FUNCTION_BLOCK "G297M_Code"	// FB 397
TITLE = G297M FAN KILN 2
//COPYRIGHT:    (C) 2009  BUHLER AG, CH-9240 UZWIL, SWITZERLAND
//
//PRODUCT:      WinCoS_BIW01_09
//
//TITLE:        FAN KILN 2
//                Machine group control
//                Maschinengruppensteuerung
// 
//--------------------------------------------------------------------------------
// 
//IDENT:        AUTHOR:             DEPT:                              DATE:
// 
//P01_FB397.2.0 M.Wedler            AEB41                              27.Apr.2010
//             2nd Release
//P01_FB397.1.0 K.Renz              CSB41                              06.Nov.2009
//             1st Release
// 
//--------------------------------------------------------------------------------
// 
//PURPOSE: 
// 
//MANUAL : 
// 
//RESTRICTIONS: 
// 
//--------------------------------------------------------------------------------
//
AUTHOR : KR
FAMILY : USW
VERSION : 9.9
VAR
  Gr : FB 10;	//Standard interface to group
  InOutValue1 : DINT ;	//Data for user
  InOutValue2 : DINT ;	//Data for user
  OutWayConflict : BOOL ;	//Data for user
  OutSelectionOk : BOOL ;	//Data for user
  CmdNewValue : BOOL ;	//Data for user
  CmdNewJob : BOOL ;	//Data for user
  OutCodeOK : BOOL ;	//Data for user
  InEndOfJob : BOOL ;	//Data for user
  staWayOk : BOOL ;	//Data for user
  EdgeStartRelease : BOOL ;	//Data for user
  USW8 : BOOL ;	//Data for user
  USW9 : BOOL ;	//Data for user
  USW10 : BOOL ;	//Data for user
  USW11 : BOOL ;	//Data for user
  USW12 : BOOL ;	//Data for user
  USW13 : BOOL ;	//Data for user
  USW14 : BOOL ;	//Data for user
  USW15 : BOOL ;	//Data for user
  A_3225_KCU04AI1 : FB 19;	// AnaInp
  A_3225_KCU04AI2 : FB 19;	// AnaInp
  A_3225_BTE05 : FB 19;	// AnaInp
  A_3225_BTE06 : FB 19;	// AnaInp
  A_3225_TSC01 : FB 14;	// DigInpCont
  A_3225_MXZ01MA : FB 1032;	// Motor+6DI
  A_3225_TSC01_AC : FB 19;	// AnaInp
  A_3225_TSC01_AF : FB 19;	// AnaInp
  A_3225_TSC01_AP : FB 19;	// AnaInp
  A_3225_TSC01_AT : FB 19;	// AnaInp
  A_3225_TSC01_COM : FB 1816;	// FU_Siemens
  A_3226_KCU04AI1 : FB 19;	// AnaInp
  A_3226_KCU04AI2 : FB 19;	// AnaInp
  A_3226_BTE05 : FB 19;	// AnaInp
  A_3226_BTE06 : FB 19;	// AnaInp
  A_3226_MXZ01MA : FB 1033;	// Motor+6DI
  A_3226_TSC01_AC : FB 19;	// AnaInp
  A_3226_TSC01_AF : FB 19;	// AnaInp
  A_3226_TSC01_AP : FB 19;	// AnaInp
  A_3226_TSC01_AT : FB 19;	// AnaInp
  A_3226_TSC01_COM : FB 1816;	// FU_Siemens
  A_3226_TSC01 : FB 14;	// DigInpCont
END_VAR
VAR_TEMP
  tmpEnable : BOOL ;
  tmpFlag : BOOL ;
  tmpCmdNext : BOOL ;
  tmpLocal : BOOL ;
  tmpAspOk : BOOL ;
  tmpHWStop : BOOL ;
  tmpInstanzDBNo : INT ;
END_VAR
BEGIN
NETWORK
TITLE =
NETWORK
TITLE = Read command from group control
//Parameter
      SET;
      S     DB9.DBX 87.0;
      R     DB9.DBX 127.0;
      R     DB9.DBX 167.0;
      R     DB9.DBX 47.0;
      R     DB9.DBX 207.0;
      S     DIX [AR2,P#32.0];
      R     DIX [AR2,P#32.1];
      R     DIX [AR2,P#32.2];
//Command
      A     DB9.DBX 327.0;
      =     DIX [AR2,P#14.0];
      A     DB9.DBX 287.0;
      =     DIX [AR2,P#15.4];
      A     DB9.DBX 407.0;
      R     DB9.DBX 407.0;
      S     DIX [AR2,P#15.3];
      A     DB9.DBX 367.0;
      R     DB9.DBX 367.0;
      S     DIX [AR2,P#15.2];
      A     DB9.DBX 447.0;
      AN    DIX [AR2,P#15.5];
      S     DIX [AR2,P#14.7];
      A     DB9.DBX 447.0;
      R     DB9.DBX 447.0;
//      U     "GCS7_GrCtrlDB".CmdManualOff[297]
//      O     "GCS7_GrCtrlDB".OutOccupied[297]
//      R     "GCS7_GrCtrlDB".CmdManualOff[297]
//      S     #Gr.CmdManualOff
      A     DB9.DBX 767.0;
      R     DB9.DBX 767.0;
      S     DIX [AR2,P#14.1];
//Init Line Number
      A     DB9.DBX 207.0;
      JCN   WE00;
      L     0;
      T     DIW [AR2,P#24.0];
WE00: NOP   0;
NETWORK
TITLE = Call Methode Control
// 1. Handle Interface PCControl      
// 2. Prepare mode --> ModePassive,ModeActive,ModeIdling      
// 3. Reset global flags of the group
      BLD   14;
      =     L 10.0;
      L     DINO;
      T     LW 8;
      CDB;
      OPN   DI [LW 8];
      TAR2  LD 4;
      L     1;
      T     DIW [AR2,P#0.0];
      +AR2  P#0.0;
      UC    FB 10;
      LAR2  LD 4;
      CDB;
      BLD   15;
NETWORK
TITLE = Restart Idling Time
      L     DIW [AR2,P#36.0];
      L     2;
      >=I;
      JC    IdTm;
      T     DIW [AR2,P#36.0];
IdTm: NOP   0;
      CLR;
      S     DIX [AR2,P#14.2];
NETWORK
TITLE = Prepare global flags
NETWORK
TITLE = Set Pattern (Target position)
      A     DIX [AR2,P#15.5];
      JC    ILO6;
// Drehzahlabsenkung wenn die andere Horde im Cooling ist
// und die Temperatur unter der eigenen Horde 5°C > als T[Soll] 
//      U     "MAL1S032Par".Par.FlagProcess.Cooling_Activ
//      U     "G302M".USW8                // Temperatur unter der Horde 5°C > T[Soll]
//      L     50                          // 50%
//      SPB   En06
      L     DB922.DBW 228;
//      U     "G275M".USW8                // Drehzahlverrinderung bei offenen Bypassklappen
//      SPBN  En06
//      L     DB799.DBW   26              // Sollwert vom LS
//      -I    
      JU    En06;
ILO6: NOP   0;
      L     DB923.DBW 284;
En06: NOP   0;
      L     100;
      *I;
      T     DIW [AR2,P#1052.0];	// xxx.xx%
      T     DIW [AR2,P#2046.0];	// xxx.xx%
NETWORK
TITLE = Interlocking WayOk
NETWORK
TITLE = Interlocking Autostart
      CLR;
      R     DIX [AR2,P#18.4];
NETWORK
TITLE = Interlocking Enable
// (network holds code this reader does not know; not shown)
//--------------------- Ein-Hordenbetrieb ----------------------------//
// Luft-Eintritt
// Luft-Austritt
//---------------------- Zwei-Hordenbetrieb --------------------------//
// Luft-Eintritt
//MW 2010.04.29      U     "G273M".A_3135_MXZ11.StHN   // Louver Air Heater Kilningbox 1
//MW 2010.04.29      U     "G299M".A_3236_MXZ11.StHN   // Recycling Air Flap Kilningbox 2
// Luft-Austritt
//MW 2010.04.29      U     "G299M".A_3235_MXZ11.StHN   // Recycling Air Flap Kilningbox 2
//MW 2010.04.29      UN    "G299M".A_3236_MXZ11.StLN   // Recycling Air Flap Kilningbox 2
//MW 2010.04.29      UN    "G273M".A_3136_MXZ11.StLN   // Recycling Air Flap Kilningbox 1
// 100% Umluft-Betrieb
//MW 2010.04.29      U     "G299M".A_3235_MXZ11.StHN   // Recycling Air Flap Kilningbox 2
//MW 2010.04.29      O     "G273M".A_3136_MXZ11.StHN   // Recycling Air Flap Kilningbox 1
//MW 2010.04.29      O     "G299M".A_3236_MXZ11.StHN   // Recycling Air Flap Kilningbox 2
NETWORK
TITLE = Interlocking Next
      A     DIX [AR2,P#15.2];
      A     DIX [AR2,P#18.4];
      AN    DIX [AR2,P#19.6];
      =     #tmpCmdNext;
NETWORK
TITLE = Interlocking Local / HWStop
      A     DB50.DBX 32.4;
      =     #tmpHWStop;
      A     DIX [AR2,P#16.0];
      O     #tmpHWStop;
      =     #tmpLocal;
NETWORK
TITLE = Interlocking Start Warning
      NOP   0;
//- Restart after fault --
      A     DIX [AR2,P#15.3];
      A     DIX [AR2,P#19.2];
      S     DB100.DBX 136.4;
//- Run Timer --
      OPN   "G297M";
      CALL  FB 100 , DB 100 (
           DIX 0.0                  := FALSE,
           DIW 2                    := 11,
           DIX 4.0                  := DBX [AR2,P#18.0],
           DIX 4.1                  := #tmpLocal,
           DIX 4.2                  := DBX [AR2,P#19.1],
           DIX 4.3                  := #tmpCmdNext,
           DIX 6.0                  := #tmpCmdNext,
           DIX 6.1                  := DBX [AR2,P#19.3]);
//- Store Startwarning done  --
//- Reset Autostart --
      A     DB100.DBX 236.1;
      FN    DIX [AR2,P#58.7];
      A     DIX [AR2,P#19.2];
      R     DIX [AR2,P#18.4];
NETWORK
TITLE = =A-3225-KCU04AI1 : VIBRATION MONITOR FAN 1 CHANNEL 1
//Alarm Level = 10.00mm/sec
//Trip Level = 11.20mm/sec
      NOP   0;
//-InLocal---
      A     #tmpLocal;
      O     DB923.DBX 1569.0;	// emergency regime without fan 1
      =     DIX [AR2,P#63.4];
//-Monitoring--- 
      CLR;
      =     DIX [AR2,P#62.0];
      CLR;
      =     DIX [AR2,P#62.1];
      CLR;
      =     DIX [AR2,P#62.2];
      SET;
      =     DIX [AR2,P#62.3];
      SET;
      =     DIX [AR2,P#62.4];
// 
//-Read inputs---
      L     PIW 1054;
      L     0;
      <I;
      JC    v003;
      TAK;
v003: T     DIW [AR2,P#66.0];
      A     DB50.DBX 32.4;
      =     DIX [AR2,P#63.0];
      A     DB51.DBX 12.5;
      =     DIX [AR2,P#63.1];
// 
//-Set Parameters---
// --> Erläuterung
      L     L#2540;	// 20mA = 25.40mm/sec       
      T     DB397.DBD 90;
      L     L#10000;	// OutValuePc=OutValueUnits
      T     DB397.DBD 94;
      L     L#-1;	// -0.01mm/sec
      T     DB397.DBD 98;
      L     L#0;	// 0.00mm/sec
      T     DB397.DBD 102;
      L     L#1000;	// 10.00mm/sec
      T     DB397.DBD 106;
      L     L#1120;	// 11.20mm/sec
      T     DB397.DBD 110;
      SET;
      =     DB397.DBX 84.6;
      =     DB397.DBX 84.7;
      =     DB397.DBX 85.0;
      =     DB397.DBX 85.1;
      =     DB397.DBX 85.6;
      =     DB397.DBX 85.7;
      CLR;
      =     DB397.DBX 85.2;
// 
//-Call object control---
      BLD   14;
// 
//-Write outputs---
      =     L 10.0;
      L     DINO;
      T     LW 8;
      CDB;
      OPN   DI [LW 8];
      TAR2  LD 4;
      +AR2  P#60.0;
      UC    FB 19;
      LAR2  LD 4;
      CDB;
      BLD   15;
NETWORK
TITLE = =A-3225-KCU04AI2 : VIBRATION MONITOR FAN 1 CHANNEL 2
//Alarm Level = 10.00mm/sec
//Trip Level = 11.20mm/sec
      NOP   0;
//-InLocal---
      A     #tmpLocal;
      O     DB923.DBX 1569.0;	// emergency regime without fan 1
      =     DIX [AR2,P#151.4];
//-Monitoring--- 
      CLR;
      =     DIX [AR2,P#150.0];
      CLR;
      =     DIX [AR2,P#150.1];
      CLR;
      =     DIX [AR2,P#150.2];
      SET;
      =     DIX [AR2,P#150.3];
      SET;
      =     DIX [AR2,P#150.4];
// 
//-Read inputs---
      L     PIW 1052;
      L     0;
      <I;
      JC    v004;
      TAK;
v004: T     DIW [AR2,P#154.0];
      A     DB50.DBX 32.4;
      =     DIX [AR2,P#151.0];
      A     DB51.DBX 12.5;
      =     DIX [AR2,P#151.1];
// 
//-Set Parameters---
// --> Erläuterung
      L     L#2540;	// 20mA = 25.40mm/sec       
      T     DB397.DBD 178;
      L     L#10000;	// OutValuePc=OutValueUnits
      T     DB397.DBD 182;
      L     L#-1;	// -0.01mm/sec
      T     DB397.DBD 186;
      L     L#0;	// 0.00mm/sec
      T     DB397.DBD 190;
      L     L#1000;	// 10.00mm/sec
      T     DB397.DBD 194;
      L     L#1120;	// 11.20mm/sec
      T     DB397.DBD 198;
      SET;
      =     DB397.DBX 172.6;
      =     DB397.DBX 172.7;
      =     DB397.DBX 173.0;
      =     DB397.DBX 173.1;
      =     DB397.DBX 173.6;
      =     DB397.DBX 173.7;
      CLR;
      =     DB397.DBX 173.2;
// 
//-Call object control---
      BLD   14;
// 
//-Write outputs---
      =     L 10.0;
      L     DINO;
      T     LW 8;
      CDB;
      OPN   DI [LW 8];
      TAR2  LD 4;
      +AR2  P#148.0;
      UC    FB 19;
      LAR2  LD 4;
      CDB;
      BLD   15;
NETWORK
TITLE = =A-3225-BTE05 : TEMPERATURE BEARING TEMPERATUR SENSOR
//Alarm Level = 100.00°C    
//Trip Level = 110.00°C
      NOP   0;
//-InLocal---
      A     #tmpLocal;
      O     DB923.DBX 1569.0;	// emergency regime without fan 1
      =     DIX [AR2,P#239.4];
//-Monitoring--- 
      CLR;
      =     DIX [AR2,P#238.0];
      CLR;
      =     DIX [AR2,P#238.1];
      CLR;
      =     DIX [AR2,P#238.2];
      SET;
      =     DIX [AR2,P#238.3];
      SET;
      =     DIX [AR2,P#238.4];
// 
//-Read inputs---
      L     PIW 1028;
      T     DIW [AR2,P#242.0];
      A     DB50.DBX 32.4;
      =     DIX [AR2,P#239.0];
      A     DB51.DBX 12.5;
      =     DIX [AR2,P#239.1];
//To Block Problems with Sensor
      L     600;
      T     DB397.DBW 296;
      T     DB397.DBW 298;
// 
//-Set Parameters---
// --> Erläuterung
      L     L#27648;	// Temperature direkt      
      T     DB397.DBD 266;
      L     L#10000;	// OutValuePc=OutValueUnits
      T     DB397.DBD 270;
      L     L#0;	// 0.00°C
      T     DB397.DBD 274;
      L     L#100;	// 1.00°C
      T     DB397.DBD 278;
      L     L#10000;	// 100.00°C
      T     DB397.DBD 282;
      L     L#11000;	// 110.00°C
      T     DB397.DBD 286;
      SET;
      =     DB397.DBX 260.6;
      =     DB397.DBX 260.7;
      =     DB397.DBX 261.0;
      =     DB397.DBX 261.1;
      =     DB397.DBX 261.6;
      =     DB397.DBX 261.7;
      CLR;
      =     DB397.DBX 261.2;
// 
//-Call object control---
      BLD   14;
// 
//-Write outputs---
      =     L 10.0;
      L     DINO;
      T     LW 8;
      CDB;
      OPN   DI [LW 8];
      TAR2  LD 4;
      +AR2  P#236.0;
      UC    FB 19;
      LAR2  LD 4;
      CDB;
      BLD   15;
NETWORK
TITLE = =A-3225-BTE06 : TEMPERATURE BEARING TEMPERATUR SENSOR
//Alarm Level = 100.00°C    
//Trip Level = 110.00°C
      NOP   0;
//-InLocal---
      A     #tmpLocal;
      O     DB923.DBX 1569.0;	// emergency regime without fan 1
      =     DIX [AR2,P#327.4];
//-Monitoring--- 
      SET;
      =     DIX [AR2,P#326.0];
      CLR;
      =     DIX [AR2,P#326.1];
      CLR;
      =     DIX [AR2,P#326.2];
      SET;
      =     DIX [AR2,P#326.3];
      SET;
      =     DIX [AR2,P#326.4];
// 
//-Read inputs---
      L     PIW 1030;
      T     DIW [AR2,P#330.0];
      A     DB50.DBX 32.4;
      =     DIX [AR2,P#327.0];
      A     DB51.DBX 12.5;
      =     DIX [AR2,P#327.1];
//To Block Problems with Sensor
      L     600;
      T     DB397.DBW 384;
      T     DB397.DBW 386;
// 
//-Set Parameters---
// --> Erläuterung
      L     L#27648;	// Temperature direkt      
      T     DB397.DBD 354;
      L     L#10000;	// OutValuePc=OutValueUnits
      T     DB397.DBD 358;
      L     L#0;	// 0.00°C
      T     DB397.DBD 362;
      L     L#100;	// 1.00°C
      T     DB397.DBD 366;
      L     L#10000;	// 100.00°C
      T     DB397.DBD 370;
      L     L#11000;	// 110.00°C
      T     DB397.DBD 374;
      SET;
      =     DB397.DBX 348.6;
      =     DB397.DBX 348.7;
      =     DB397.DBX 349.0;
      =     DB397.DBX 349.1;
      =     DB397.DBX 349.6;
      =     DB397.DBX 349.7;
      CLR;
      =     DB397.DBX 349.2;
// 
//-Call object control---
      BLD   14;
// 
//-Write outputs---
      =     L 10.0;
      L     DINO;
      T     LW 8;
      CDB;
      OPN   DI [LW 8];
      TAR2  LD 4;
      +AR2  P#324.0;
      UC    FB 19;
      LAR2  LD 4;
      CDB;
      BLD   15;
NETWORK
TITLE = =A-3225-MXZ01MA : FAN 1
      NOP   0;
//-InLocal---
      A     #tmpLocal;
      O     DB923.DBX 1569.0;	// emergency regime without fan 1
      =     DIX [AR2,P#449.4];
//-Interlocking---
      AN    DB923.DBX 1569.0;	// emergency regime without fan 1
      A(;
      AN    DIX [AR2,P#1445.4];
      O     DB923.DBX 1569.1;	// emergency regime without fan 2
      );
      A(;
      A     DIX [AR2,P#15.5];
      A     DIX [AR2,P#14.5];
      ON    DIX [AR2,P#15.5];
      );
      AN    DIX [AR2,P#65.7];	// Vibrationswächter 1
      AN    DIX [AR2,P#153.7];	// Vibrationswächter 2
      AN    DIX [AR2,P#241.7];	// Lager Temperatur 1
      AN    DIX [AR2,P#329.7];	// Lager Temperatur 2
      AN    DB376.DBX 65.4;	// Differenzdruck hinter dem Waermetauscher
      A     DIX [AR2,P#18.0];
      =     DIX [AR2,P#448.1];
      A     #tmpCmdNext;
//      U     "MAL1S033Par".Par.FlagProcess2.Schaltp_5
      S     DIX [AR2,P#449.2];
      A     DIX [AR2,P#19.7];
      =     DIX [AR2,P#449.7];
// 
//=Values and commands of elements===
//-=A-3225-KCU04---
//      CLR
//      S     #A_3225_MXZ01MA.A_3225_KCU04.CmdRunTimeOutTime
//-=A-3225-MXZ01_SM---
//      CLR
//      S     #A_3225_MXZ01MA.A_3225_MXZ01_SM.CmdRunTimeOutTime
// 
//-Read inputs of elements---
      O     DIX [AR2,P#451.1];
      O     DIX [AR2,P#451.2];
      =     DIX [AR2,P#494.6];
      A     I 1026.6;
      =     DIX [AR2,P#460.6];
      A     DB50.DBX 32.4;
      =     DIX [AR2,P#462.0];
      A     DB51.DBX 12.6;
      =     DIX [AR2,P#462.1];
      A     DB50.DBX 32.4;
      =     DIX [AR2,P#496.0];
      A     DIX [AR2,P#1050.4];
      O     DB50.DBX 33.0;
      A     DIX [AR2,P#666.6];
      =     DIX [AR2,P#664.6];
      A     DB50.DBX 32.4;
      =     DIX [AR2,P#666.0];
// Überwachung Profibus-Kommunikation
      A     DB51.DBX 12.7;	// FU  ?????
      =     DIX [AR2,P#666.1];
// 
//-Set Parameters---
// 
//-Call object control---
      BLD   14;
// 
//-Write outputs---
      =     L 10.0;
      L     DINO;
      T     LW 8;
      CDB;
      OPN   DI [LW 8];
      TAR2  LD 4;
      +AR2  P#446.0;
      UC    "A_3225_MXZ01MA_Code";
      LAR2  LD 4;
      CDB;
      BLD   15;
NETWORK
TITLE = =A-3225-TSC01_COM : FAN 1 FU KOMMUNIKATION
      NOP   0;
      A     DIX [AR2,P#666.6];
      =     DIX [AR2,P#1050.1];
//      U     #A_3225_MXZ01MA.A_3225_MXZ01.OutpRunRev
      CLR;
      =     DIX [AR2,P#1050.0];
      A     DIX [AR2,P#15.3];
      O     DIX [AR2,P#462.6];
      S     DIX [AR2,P#1050.2];
// 
//-Read inputs---
// 
//-Set Parameters---
// 
//-Call object control---
      BLD   14;
// 
//-Write outputs---
      =     L 10.0;
      L     DINO;
      T     LW 8;
      CDB;
      OPN   DI [LW 8];
      TAR2  LD 4;
      +AR2  P#1048.0;
      UC    FB 1816;
      LAR2  LD 4;
      CDB;
      BLD   15;
NETWORK
TITLE = =A-3225-TSC01_AC : ACT. CURRENT FAN 1 FU 
//20000Dez=100,0%=720,0A
//Analog Input 20mA=27648Dez=995,3A
      NOP   0;
//-InLocal---
      A     #tmpLocal;
      O     DB923.DBX 1569.0;	// emergency regime without fan 1
      =     DIX [AR2,P#699.4];
//-Monitoring--- 
      SET;
      =     DIX [AR2,P#698.0];
      CLR;
      =     DIX [AR2,P#698.1];
      CLR;
      =     DIX [AR2,P#698.2];
      CLR;
      =     DIX [AR2,P#698.3];
      CLR;
      =     DIX [AR2,P#698.4];
// 
//-Read inputs---
      L     DIW [AR2,P#1058.0];
      T     DIW [AR2,P#702.0];
      A     DB50.DBX 32.4;
      =     DIX [AR2,P#699.0];
// 
//-Set Parameters---
// --> Erläuterung
      L     L#9953;	// Stromwert bei 27648Dez
      T     DB397.DBD 726;
      L     L#10000;	// OutValuePc=OutValueUnits
      T     DB397.DBD 730;
      L     L#0;	// 0.0A
      T     DB397.DBD 734;
      L     L#4000;	// 40.0A
      T     DB397.DBD 738;
      L     L#7200;	// 720.0A=100.0%
      T     DB397.DBD 742;
      L     L#9360;	// 936.0A=130.0%
      T     DB397.DBD 746;
// 
//-Call object control---
      BLD   14;
// 
//-Write outputs---
      =     L 10.0;
      L     DINO;
      T     LW 8;
      CDB;
      OPN   DI [LW 8];
      TAR2  LD 4;
      +AR2  P#696.0;
      UC    FB 19;
      LAR2  LD 4;
      CDB;
      BLD   15;
NETWORK
TITLE = =A-3225-TSC01_AF : ACT. FREQUENCY FAN 1 FU 
      NOP   0;
//-InLocal---
      A     #tmpLocal;
      O     DB923.DBX 1569.0;	// emergency regime without fan 1
      =     DIX [AR2,P#787.4];
//-Monitoring--- 
      SET;
      =     DIX [AR2,P#786.0];
      CLR;
      =     DIX [AR2,P#786.1];
      CLR;
      =     DIX [AR2,P#786.2];
      CLR;
      =     DIX [AR2,P#786.3];
      CLR;
      =     DIX [AR2,P#786.4];
// 
//-Read inputs---
      L     DIW [AR2,P#1048.0];	// Umgerechnet in FU-FB
      T     DIW [AR2,P#790.0];
      A     DB50.DBX 32.4;
      =     DIX [AR2,P#787.0];
// 
//-Set Parameters---
// --> Erläuterung
      L     L#27648;	// InpValue=Drehzahl direkt   
      T     DB397.DBD 814;
      L     L#10000;	// OutValuePc=OutValueUnits
      T     DB397.DBD 818;
      L     L#4000;	// 40.00% ist untere Grenze
      T     DB397.DBD 822;
      L     L#4100;	// 41.00%
      T     DB397.DBD 826;
      L     L#8000;	// 80.00%
      T     DB397.DBD 830;
      L     L#10100;	// 101.00%
      T     DB397.DBD 834;
// 
//-Call object control---
      BLD   14;
// 
//-Write outputs---
      =     L 10.0;
      L     DINO;
      T     LW 8;
      CDB;
      OPN   DI [LW 8];
      TAR2  LD 4;
      +AR2  P#784.0;
      UC    FB 19;
      LAR2  LD 4;
      CDB;
      BLD   15;
NETWORK
TITLE = =A-3225-TSC01_AP : ACT. POWER FAN 1 FU 
      NOP   0;
//-InLocal---
      A     #tmpLocal;
      O     DB923.DBX 1569.0;	// emergency regime without fan 1
      =     DIX [AR2,P#875.4];
//-Monitoring--- 
      CLR;
      =     DIX [AR2,P#874.0];
      CLR;
      =     DIX [AR2,P#874.1];
      CLR;
      =     DIX [AR2,P#874.2];
      CLR;
      =     DIX [AR2,P#874.3];
      CLR;
      =     DIX [AR2,P#874.4];
// 
//-Read inputs---
      L     DIW [AR2,P#1060.0];
      T     DIW [AR2,P#878.0];
      A     DB50.DBX 32.4;
      =     DIX [AR2,P#875.0];
// 
//-Set Parameters---
// 
//-Call object control---
      BLD   14;
// 
//-Write outputs---
      =     L 10.0;
      L     DINO;
      T     LW 8;
      CDB;
      OPN   DI [LW 8];
      TAR2  LD 4;
      +AR2  P#872.0;
      UC    FB 19;
      LAR2  LD 4;
      CDB;
      BLD   15;
NETWORK
TITLE = =A-3225-TSC01_AT : ACT. TORQUE FAN 1 FU 
      NOP   0;
//-InLocal---
      A     #tmpLocal;
      O     DB923.DBX 1569.0;	// emergency regime without fan 1
      =     DIX [AR2,P#963.4];
//-Monitoring--- 
      CLR;
      =     DIX [AR2,P#962.0];
      CLR;
      =     DIX [AR2,P#962.1];
      CLR;
      =     DIX [AR2,P#962.2];
      CLR;
      =     DIX [AR2,P#962.3];
      CLR;
      =     DIX [AR2,P#962.4];
// 
//-Read inputs---
      L     DIW [AR2,P#1062.0];
      T     DIW [AR2,P#966.0];
      A     DB50.DBX 32.4;
      =     DIX [AR2,P#963.0];
// 
//-Set Parameters---
// 
//-Call object control---
      BLD   14;
// 
//-Write outputs---
      =     L 10.0;
      L     DINO;
      T     LW 8;
      CDB;
      OPN   DI [LW 8];
      TAR2  LD 4;
      +AR2  P#960.0;
      UC    FB 19;
      LAR2  LD 4;
      CDB;
      BLD   15;
NETWORK
TITLE = =A-3226-KCU04AI1 : VIBRATION MONITOR FAN 2 CHANNEL 1
//Alarm Level = 10.00mm/sec
//Trip Level = 11.20mm/sec
      NOP   0;
//-InLocal---
      A     #tmpLocal;
      O     DB923.DBX 1569.1;	// emergency regime without fan 2
      =     DIX [AR2,P#1091.4];
//-Monitoring--- 
      CLR;
      =     DIX [AR2,P#1090.0];
      CLR;
      =     DIX [AR2,P#1090.1];
      CLR;
      =     DIX [AR2,P#1090.2];
      SET;
      =     DIX [AR2,P#1090.3];
      SET;
      =     DIX [AR2,P#1090.4];
// 
//-Read inputs---
      L     PIW 1058;
      L     0;
      <I;
      JC    v013;
      TAK;
v013: T     DIW [AR2,P#1094.0];
      A     DB50.DBX 32.4;
      =     DIX [AR2,P#1091.0];
      A     DB51.DBX 12.5;
      =     DIX [AR2,P#1091.1];
// 
//-Set Parameters---
// --> Erläuterung
      L     L#2540;	// 20mA = 25.40mm/sec       
      T     DB397.DBD 1118;
      L     L#10000;	// OutValuePc=OutValueUnits
      T     DB397.DBD 1122;
      L     L#-1;	// -0.01mm/sec
      T     DB397.DBD 1126;
      L     L#0;	// 0.00mm/sec
      T     DB397.DBD 1130;
      L     L#1000;	// 10.00mm/sec
      T     DB397.DBD 1134;
      L     L#1120;	// 11.20mm/sec
      T     DB397.DBD 1138;
      SET;
      =     DB397.DBX 1112.6;
      =     DB397.DBX 1112.7;
      =     DB397.DBX 1113.0;
      =     DB397.DBX 1113.1;
      =     DB397.DBX 1113.6;
      =     DB397.DBX 1113.7;
      CLR;
      =     DB397.DBX 1113.2;
// 
//-Call object control---
      BLD   14;
// 
//-Write outputs---
      =     L 10.0;
      L     DINO;
      T     LW 8;
      CDB;
      OPN   DI [LW 8];
      TAR2  LD 4;
      +AR2  P#1088.0;
      UC    FB 19;
      LAR2  LD 4;
      CDB;
      BLD   15;
NETWORK
TITLE = =A-3226-KCU04AI2 : VIBRATION MONITOR FAN 2 CHANNEL 2
//Alarm Level = 10.00mm/sec
//Trip Level = 11.20mm/sec
      NOP   0;
//-InLocal---
      A     #tmpLocal;
      O     DB923.DBX 1569.1;	// emergency regime without fan 2
      =     DIX [AR2,P#1179.4];
//-Monitoring--- 
      CLR;
      =     DIX [AR2,P#1178.0];
      CLR;
      =     DIX [AR2,P#1178.1];
      CLR;
      =     DIX [AR2,P#1178.2];
      SET;
      =     DIX [AR2,P#1178.3];
      SET;
      =     DIX [AR2,P#1178.4];
// 
//-Read inputs---
      L     PIW 1056;
      L     0;
      <I;
      JC    v014;
      TAK;
v014: T     DIW [AR2,P#1182.0];
      A     DB50.DBX 32.4;
      =     DIX [AR2,P#1179.0];
      A     DB51.DBX 12.5;
      =     DIX [AR2,P#1179.1];
// 
//-Set Parameters---
// --> Erläuterung
      L     L#2540;	// 20mA = 25.40mm/sec       
      T     DB397.DBD 1206;
      L     L#10000;	// OutValuePc=OutValueUnits
      T     DB397.DBD 1210;
      L     L#-1;	// -0.01mm/sec
      T     DB397.DBD 1214;
      L     L#0;	// 0.00mm/sec
      T     DB397.DBD 1218;
      L     L#1000;	// 10.00mm/sec
      T     DB397.DBD 1222;
      L     L#1120;	// 11.20mm/sec
      T     DB397.DBD 1226;
      SET;
      =     DB397.DBX 1200.6;
      =     DB397.DBX 1200.7;
      =     DB397.DBX 1201.0;
      =     DB397.DBX 1201.1;
      =     DB397.DBX 1201.6;
      =     DB397.DBX 1201.7;
      CLR;
      =     DB397.DBX 1201.2;
// 
//-Call object control---
      BLD   14;
// 
//-Write outputs---
      =     L 10.0;
      L     DINO;
      T     LW 8;
      CDB;
      OPN   DI [LW 8];
      TAR2  LD 4;
      +AR2  P#1176.0;
      UC    FB 19;
      LAR2  LD 4;
      CDB;
      BLD   15;
NETWORK
TITLE = =A-3226-BTE05 : TEMPERATURE BEARING TEMPERATUR SENSOR
//Alarm Level = 100.00°C    
//Trip Level = 110.00°C
      NOP   0;
//-InLocal---
      A     #tmpLocal;
      O     DB923.DBX 1569.1;	// emergency regime without fan 2
      =     DIX [AR2,P#1267.4];
//-Monitoring--- 
      CLR;
      =     DIX [AR2,P#1266.0];
      CLR;
      =     DIX [AR2,P#1266.1];
      CLR;
      =     DIX [AR2,P#1266.2];
      SET;
      =     DIX [AR2,P#1266.3];
      SET;
      =     DIX [AR2,P#1266.4];
// 
//-Read inputs---
      L     PIW 1032;
      T     DIW [AR2,P#1270.0];
      A     DB50.DBX 32.4;
      =     DIX [AR2,P#1267.0];
      A     DB51.DBX 12.5;
      =     DIX [AR2,P#1267.1];
//To Block Problems with Sensor
      L     600;
      T     DB397.DBW 1324;
      T     DB397.DBW 1326;
// 
//-Set Parameters---
// --> Erläuterung
      L     L#27648;	// Temperature direkt      
      T     DB397.DBD 1294;
      L     L#10000;	// OutValuePc=OutValueUnits
      T     DB397.DBD 1298;
      L     L#0;	// 0.00°C
      T     DB397.DBD 1302;
      L     L#100;	// 1.00°C
      T     DB397.DBD 1306;
      L     L#10000;	// 100.00°C
      T     DB397.DBD 1310;
      L     L#11000;	// 110.00°C
      T     DB397.DBD 1314;
      SET;
      =     DB397.DBX 1288.6;
      =     DB397.DBX 1288.7;
      =     DB397.DBX 1289.0;
      =     DB397.DBX 1289.1;
      =     DB397.DBX 1289.6;
      =     DB397.DBX 1289.7;
      CLR;
      =     DB397.DBX 1289.2;
// 
//-Call object control---
      BLD   14;
// 
//-Write outputs---
      =     L 10.0;
      L     DINO;
      T     LW 8;
      CDB;
      OPN   DI [LW 8];
      TAR2  LD 4;
      +AR2  P#1264.0;
      UC    FB 19;
      LAR2  LD 4;
      CDB;
      BLD   15;
NETWORK
TITLE = =A-3226-BTE06 : TEMPERATURE BEARING TEMPERATUR SENSOR
//Alarm Level = 100.00°C    
//Trip Level = 110.00°C
      NOP   0;
//-InLocal---
      A     #tmpLocal;
      O     DB923.DBX 1569.1;	// emergency regime without fan 2
      =     DIX [AR2,P#1355.4];
//-Monitoring--- 
      CLR;
      =     DIX [AR2,P#1354.0];
      CLR;
      =     DIX [AR2,P#1354.1];
      CLR;
      =     DIX [AR2,P#1354.2];
      SET;
      =     DIX [AR2,P#1354.3];
      SET;
      =     DIX [AR2,P#1354.4];
// 
//-Read inputs---
      L     PIW 1034;
      T     DIW [AR2,P#1358.0];
      A     DB50.DBX 32.4;
      =     DIX [AR2,P#1355.0];
      A     DB51.DBX 12.5;
      =     DIX [AR2,P#1355.1];
//To Block Problems with Sensor
      L     600;
      T     DB397.DBW 1412;
      T     DB397.DBW 1414;
// 
//-Set Parameters---
// --> Erläuterung
      L     L#27648;	// Temperature direkt      
      T     DB397.DBD 1382;
      L     L#10000;	// OutValuePc=OutValueUnits
      T     DB397.DBD 1386;
      L     L#0;	// 0.00°C
      T     DB397.DBD 1390;
      L     L#100;	// 1.00°C
      T     DB397.DBD 1394;
      L     L#10000;	// 100.00°C
      T     DB397.DBD 1398;
      L     L#11000;	// 110.00°C
      T     DB397.DBD 1402;
      SET;
      =     DB397.DBX 1376.6;
      =     DB397.DBX 1376.7;
      =     DB397.DBX 1377.0;
      =     DB397.DBX 1377.1;
      =     DB397.DBX 1377.6;
      =     DB397.DBX 1377.7;
      CLR;
      =     DB397.DBX 1377.2;
// 
//-Call object control---
      BLD   14;
// 
//-Write outputs---
      =     L 10.0;
      L     DINO;
      T     LW 8;
      CDB;
      OPN   DI [LW 8];
      TAR2  LD 4;
      +AR2  P#1352.0;
      UC    FB 19;
      LAR2  LD 4;
      CDB;
      BLD   15;
NETWORK
TITLE = =A-3226-MXZ01MA : FAN 2
      NOP   0;
//-InLocal---
      A     #tmpLocal;
      O     DB923.DBX 1569.1;	// emergency regime without fan 2
      =     DIX [AR2,P#1443.4];
//-Interlocking---
      AN    DB923.DBX 1569.1;	// emergency regime without fan 2
      A(;
      AN    DIX [AR2,P#451.4];
      O     DB923.DBX 1569.0;	// emergency regime without fan 1
      );
      A(;
      A     DIX [AR2,P#15.5];
      A     DIX [AR2,P#14.5];
      ON    DIX [AR2,P#15.5];
      );
      AN    DIX [AR2,P#1093.7];	// Vibrationswächter 1
      AN    DIX [AR2,P#1181.7];	// Vibrationswächter 2
      AN    DIX [AR2,P#1269.7];	// Lager Temperatur 1
      AN    DIX [AR2,P#1357.7];	// Lager Temperatur 2
      AN    DB376.DBX 65.4;	// Differenzdruck hinter dem Waermetauscher
      A     DIX [AR2,P#18.0];
      =     DIX [AR2,P#1442.1];
      A     #tmpCmdNext;
//      U     "MAL1S033Par".Par.FlagProcess2.Schaltp_5
      S     DIX [AR2,P#1443.2];
      A     DIX [AR2,P#19.7];
      =     DIX [AR2,P#1443.7];
// 
//=Values and commands of elements===
//-=A-3226-KCU04---
//      CLR
//      S     #A_3226_MXZ01MA.A_3226_KCU04.CmdRunTimeOutTime
//-=A-3226-MXZ01_SM---
//      CLR
//      S     #A_3226_MXZ01MA.A_3226_MXZ01_SM.CmdRunTimeOutTime
// 
//-Read inputs of elements---
      O     DIX [AR2,P#1445.1];
      O     DIX [AR2,P#1445.2];
      =     DIX [AR2,P#1488.6];
      A     I 1026.7;
      =     DIX [AR2,P#1454.6];
      A     DB50.DBX 32.4;
      =     DIX [AR2,P#1456.0];
      A     DB51.DBX 12.6;
      =     DIX [AR2,P#1456.1];
      A     DB50.DBX 32.4;
      =     DIX [AR2,P#1490.0];
      A     DIX [AR2,P#2044.4];
      O     DB50.DBX 33.0;
      A     DIX [AR2,P#1660.6];
      =     DIX [AR2,P#1658.6];
      A     DB50.DBX 32.4;
      =     DIX [AR2,P#1660.0];
// Überwachung Profibus-Kommunikation
      A     DB51.DBX 13.0;	// FU  ?????
      =     DIX [AR2,P#1660.1];
// 
//-Set Parameters---
// 
//-Call object control---
      BLD   14;
// 
//-Write outputs---
      =     L 10.0;
      L     DINO;
      T     LW 8;
      CDB;
      OPN   DI [LW 8];
      TAR2  LD 4;
      +AR2  P#1440.0;
      UC    "A_3226_MXZ01MA_Code";
      LAR2  LD 4;
      CDB;
      BLD   15;
NETWORK
TITLE = =A-3226-TSC01_COM : FAN 2 FU KOMMUNIKATION
      NOP   0;
      A     DIX [AR2,P#1660.6];
      =     DIX [AR2,P#2044.1];
//      U     #A_3226_MXZ01MA.A_3226_MXZ01.OutpRunRev
      CLR;
      =     DIX [AR2,P#2044.0];
      A     DIX [AR2,P#15.3];
      O     DIX [AR2,P#1456.6];
      S     DIX [AR2,P#2044.2];
// 
//-Read inputs---
// 
//-Set Parameters---
// 
//-Call object control---
      BLD   14;
// 
//-Write outputs---
      =     L 10.0;
      L     DINO;
      T     LW 8;
      CDB;
      OPN   DI [LW 8];
      TAR2  LD 4;
      +AR2  P#2042.0;
      UC    FB 1816;
      LAR2  LD 4;
      CDB;
      BLD   15;
NETWORK
TITLE = =A-3226-TSC01_AC : ACT. CURRENT FAN 2 FU 
//20000Dez=100,0%=720,0A
//Analog Input 20mA=27648Dez=995,3A
      NOP   0;
//-InLocal---
      A     #tmpLocal;
      O     DB923.DBX 1569.1;	// emergency regime without fan 2
      =     DIX [AR2,P#1693.4];
//-Monitoring--- 
      CLR;
      =     DIX [AR2,P#1692.0];
      CLR;
      =     DIX [AR2,P#1692.1];
      CLR;
      =     DIX [AR2,P#1692.2];
      CLR;
      =     DIX [AR2,P#1692.3];
      CLR;
      =     DIX [AR2,P#1692.4];
// 
//-Read inputs---
      L     DIW [AR2,P#2052.0];
      T     DIW [AR2,P#1696.0];
      A     DB50.DBX 32.4;
      =     DIX [AR2,P#1693.0];
// 
//-Set Parameters---
      L     L#9953;	// Stromwert bei 27648Dez
      T     DB397.DBD 1720;
      L     L#10000;	// OutValuePc=OutValueUnits
      T     DB397.DBD 1724;
      L     L#0;	// 0.0A
      T     DB397.DBD 1728;
      L     L#4000;	// 40.0A
      T     DB397.DBD 1732;
      L     L#7200;	// 720.0A=100.0%
      T     DB397.DBD 1736;
      L     L#9360;	// 936.0A=130.0%
      T     DB397.DBD 1740;
// 
//-Call object control---
      BLD   14;
// 
//-Write outputs---
      =     L 10.0;
      L     DINO;
      T     LW 8;
      CDB;
      OPN   DI [LW 8];
      TAR2  LD 4;
      +AR2  P#1690.0;
      UC    FB 19;
      LAR2  LD 4;
      CDB;
      BLD   15;
NETWORK
TITLE = =A-3226-TSC01_AF : ACT. FREQUENCY FAN 2 FU 
      NOP   0;
//-InLocal---
      A     #tmpLocal;
      O     DB923.DBX 1569.1;	// emergency regime without fan 2
      =     DIX [AR2,P#1781.4];
//-Monitoring--- 
      SET;
      =     DIX [AR2,P#1780.0];
      CLR;
      =     DIX [AR2,P#1780.1];
      CLR;
      =     DIX [AR2,P#1780.2];
      CLR;
      =     DIX [AR2,P#1780.3];
      CLR;
      =     DIX [AR2,P#1780.4];
// 
//-Read inputs---
      L     DIW [AR2,P#2042.0];	// Umgerechnet in FU-FB  
      T     DIW [AR2,P#1784.0];
      A     DB50.DBX 32.4;
      =     DIX [AR2,P#1781.0];
// 
//-Set Parameters---
// --> Erläuterung
      L     L#27648;	// InpValue=Drehzahl direkt   
      T     DB397.DBD 1808;
      L     L#10000;	// OutValuePc=OutValueUnits
      T     DB397.DBD 1812;
      L     L#4000;	// 40.00% ist untere Grenze
      T     DB397.DBD 1816;
      L     L#4100;	// 41.00%
      T     DB397.DBD 1820;
      L     L#8000;	// 80.00%
      T     DB397.DBD 1824;
      L     L#10100;	// 101.00%
      T     DB397.DBD 1828;
// 
//-Call object control---
      BLD   14;
// 
//-Write outputs---
      =     L 10.0;
      L     DINO;
      T     LW 8;
      CDB;
      OPN   DI [LW 8];
      TAR2  LD 4;
      +AR2  P#1778.0;
      UC    FB 19;
      LAR2  LD 4;
      CDB;
      BLD   15;
NETWORK
TITLE = =A-3226-TSC01_AP : ACT. POWER FAN 2 FU 
      NOP   0;
//-InLocal---
      A     #tmpLocal;
      O     DB923.DBX 1569.1;	// emergency regime without fan 2
      =     DIX [AR2,P#1869.4];
//-Monitoring--- 
      CLR;
      =     DIX [AR2,P#1868.0];
      CLR;
      =     DIX [AR2,P#1868.1];
      CLR;
      =     DIX [AR2,P#1868.2];
      CLR;
      =     DIX [AR2,P#1868.3];
      CLR;
      =     DIX [AR2,P#1868.4];
// 
//-Read inputs---
      L     DIW [AR2,P#2054.0];
      T     DIW [AR2,P#1872.0];
      A     DB50.DBX 32.4;
      =     DIX [AR2,P#1869.0];
// 
//-Set Parameters---
// 
//-Call object control---
      BLD   14;
// 
//-Write outputs---
      =     L 10.0;
      L     DINO;
      T     LW 8;
      CDB;
      OPN   DI [LW 8];
      TAR2  LD 4;
      +AR2  P#1866.0;
      UC    FB 19;
      LAR2  LD 4;
      CDB;
      BLD   15;
NETWORK
TITLE = =A-3226-TSC01_AT : ACT. TORQUE FAN 2 FU 
      NOP   0;
//-InLocal---
      A     #tmpLocal;
      O     DB923.DBX 1569.1;	// emergency regime without fan 2
      =     DIX [AR2,P#1957.4];
//-Monitoring--- 
      CLR;
      =     DIX [AR2,P#1956.0];
      CLR;
      =     DIX [AR2,P#1956.1];
      CLR;
      =     DIX [AR2,P#1956.2];
      CLR;
      =     DIX [AR2,P#1956.3];
      CLR;
      =     DIX [AR2,P#1956.4];
// 
//-Read inputs---
      L     DIW [AR2,P#2056.0];
      T     DIW [AR2,P#1960.0];
      A     DB50.DBX 32.4;
      =     DIX [AR2,P#1957.0];
// 
//-Set Parameters---
// 
//-Call object control---
      BLD   14;
// 
//-Write outputs---
      =     L 10.0;
      L     DINO;
      T     LW 8;
      CDB;
      OPN   DI [LW 8];
      TAR2  LD 4;
      +AR2  P#1954.0;
      UC    FB 19;
      LAR2  LD 4;
      CDB;
      BLD   15;
NETWORK
TITLE = =A-3225-TSC01 : FAN 1 FU KOMMUNIKATION
      NOP   0;
//-InLocal---
      A     #tmpLocal;
      =     DIX [AR2,P#415.4];
// 
//-Monitoring---
      CLR;
      =     DIX [AR2,P#414.0];
      CLR;
      =     DIX [AR2,P#414.1];
// 
//-PreAlarm---
      CLR;
      =     DIX [AR2,P#414.2];
      CLR;
      =     DIX [AR2,P#414.3];
// 
//-Additional commands---
//      CLR
//      S     #A_3225_TSC01.CmdRunTimeOutTime
// 
//-Read inputs---
      A     DIX [AR2,P#1054.1];
      A     DIX [AR2,P#1055.1];
      AN    DIX [AR2,P#1055.3];
      =     DIX [AR2,P#414.6];
// 
//-Set Parameters---
// 
//-Call object control---
      BLD   14;
// 
//-Write outputs---
      =     L 10.0;
      L     DINO;
      T     LW 8;
      CDB;
      OPN   DI [LW 8];
      TAR2  LD 4;
      +AR2  P#412.0;
      UC    FB 14;
      LAR2  LD 4;
      CDB;
      BLD   15;
NETWORK
TITLE = =A-3226-TSC01 : FAN 2 FU KOMMUNIKATION
      NOP   0;
//-InLocal---
      A     #tmpLocal;
      =     DIX [AR2,P#2085.4];
// 
//-Monitoring---
      CLR;
      =     DIX [AR2,P#2084.0];
      CLR;
      =     DIX [AR2,P#2084.1];
// 
//-PreAlarm---
      CLR;
      =     DIX [AR2,P#2084.2];
      CLR;
      =     DIX [AR2,P#2084.3];
// 
//-Additional commands---
//      CLR
//      S     #A_3226_TSC01.CmdRunTimeOutTime
// 
//-Read inputs---
      A     DIX [AR2,P#2048.1];
      A     DIX [AR2,P#2049.1];
      AN    DIX [AR2,P#2049.3];
      =     DIX [AR2,P#2084.6];
// 
//-Set Parameters---
// 
//-Call object control---
      BLD   14;
// 
//-Write outputs---
      =     L 10.0;
      L     DINO;
      T     LW 8;
      CDB;
      OPN   DI [LW 8];
      TAR2  LD 4;
      +AR2  P#2082.0;
      UC    FB 14;
      LAR2  LD 4;
      CDB;
      BLD   15;
NETWORK
TITLE = Test Fault
      A     DIX [AR2,P#65.7];
      O     DIX [AR2,P#153.7];
      O     DIX [AR2,P#241.7];
      O     DIX [AR2,P#329.7];
      O     DIX [AR2,P#451.4];
      O     DIX [AR2,P#701.7];
      O     DIX [AR2,P#789.7];
      O     DIX [AR2,P#877.7];
      O     DIX [AR2,P#965.7];
      O     DIX [AR2,P#1093.7];
      O     DIX [AR2,P#1181.7];
      O     DIX [AR2,P#1269.7];
      O     DIX [AR2,P#1357.7];
      O     DIX [AR2,P#1445.4];
      O     DIX [AR2,P#1695.7];
      O     DIX [AR2,P#1783.7];
      O     DIX [AR2,P#1871.7];
      O     DIX [AR2,P#1959.7];
      O     DIX [AR2,P#417.4];
      O     DIX [AR2,P#2087.4];
      =     DIX [AR2,P#19.2];
NETWORK
TITLE = Test Warning
      A     DIX [AR2,P#65.6];
      O     DIX [AR2,P#153.6];
      O     DIX [AR2,P#241.6];
      O     DIX [AR2,P#329.6];
      O     DIX [AR2,P#701.6];
      O     DIX [AR2,P#789.6];
      O     DIX [AR2,P#877.6];
      O     DIX [AR2,P#965.6];
      O     DIX [AR2,P#1093.6];
      O     DIX [AR2,P#1181.6];
      O     DIX [AR2,P#1269.6];
      O     DIX [AR2,P#1357.6];
      O     DIX [AR2,P#1695.6];
      O     DIX [AR2,P#1783.6];
      O     DIX [AR2,P#1871.6];
      O     DIX [AR2,P#1959.6];
      =     DIX [AR2,P#17.6];
NETWORK
TITLE = Test Stopped
      A     DIX [AR2,P#451.0];
      A     DIX [AR2,P#1445.0];
      AN    DIX [AR2,P#19.2];
      =     DIX [AR2,P#19.0];
NETWORK
TITLE = Test Started
      A(;
      A     DIX [AR2,P#451.2];
      O     DB923.DBX 1569.0;	// emergency regime without fan 1
      );
      A(;
      A     DIX [AR2,P#1445.2];
      O     DB923.DBX 1569.1;	// emergency regime without fan 2
      );
      AN    DIX [AR2,P#19.0];
      AN    DIX [AR2,P#19.2];
      =     DIX [AR2,P#19.1];
NETWORK
TITLE = Enable Previous Group
      A     DIX [AR2,P#451.2];
      A     DIX [AR2,P#788.1];	// InpValue>=ParL
      A     DIX [AR2,P#1445.2];
      A     DIX [AR2,P#1782.1];	// InpValue>=ParL
      O;
      A     DIX [AR2,P#451.2];
      A     DIX [AR2,P#788.2];	// InpValue>=ParH
      O;
      A     DIX [AR2,P#1445.2];
      A     DIX [AR2,P#1782.2];	// InpValue>=ParH
      =     DIX [AR2,P#18.7];
NETWORK
TITLE = Call Methode State
//1. Make State of the group: This function use the signals:
//        Gr.VarStopped, Gr.VarStarted, Gr.VarFault
//2.Reset Commands to group: e.g.CmdFaultReset
      BLD   14;
      =     L 10.0;
      L     DINO;
      T     LW 8;
      CDB;
      OPN   DI [LW 8];
      TAR2  LD 4;
      L     2;
      T     DIW [AR2,P#0.0];
      +AR2  P#0.0;
      UC    FB 10;
      LAR2  LD 4;
      CDB;
      BLD   15;
NETWORK
TITLE = Init
      SET;
      R     DIX [AR2,P#58.2];
      R     DIX [AR2,P#58.3];
NETWORK
TITLE = Write data to group control
      A     DIX [AR2,P#17.0];
      =     DB9.DBX 487.0;
      A     DIX [AR2,P#17.2];
      =     DB9.DBX 527.0;
      A     DIX [AR2,P#17.4];
      =     DB9.DBX 567.0;
      A     DIX [AR2,P#17.6];
      =     DB9.DBX 607.0;
      A     DIX [AR2,P#18.5];
      =     DB9.DBX 647.0;
      A     DIX [AR2,P#18.2];
      =     DB9.DBX 887.0;
      A     DIX [AR2,P#18.3];
      =     DB9.DBX 847.0;
      A     DIX [AR2,P#17.5];
      =     DB9.DBX 807.0;
      A     DIX [AR2,P#18.4];
      =     DB9.DBX 927.0;
      A     DIX [AR2,P#19.3];
      =     DB9.DBX 967.0;
NETWORK
TITLE = End of block
      BE;
END_FUNCTION_BLOCK

FUNCTION_BLOCK "A_3125_MXZ01MA_Code"	// FB 1018
TITLE = A_3125_MXZ01MA FAN 1
//COPYRIGHT:     (C) 2009  BUHLER AG, CH-9240 UZWIL, SWITZERLAND
//
//PRODUCT:       WinCoS_BIW01_09
//
//TITLE:         FAN 1
// 
//--------------------------------------------------------------------------------
// 
//IDENT:         AUTHOR:             DEPT:                             DATE:
// 
//P01_FB1018.1.0 K.Renz              CSB41                             07.Okt.2009
//               1st Release
// 
//--------------------------------------------------------------------------------
// 
//PURPOSE: 
// 
//MANUAL : 
// 
//RESTRICTIONS: 
// 
//--------------------------------------------------------------------------------
//
AUTHOR : KR
FAMILY : USW
VERSION : 0.0
VAR
  Ma : UDT 20500;	// Machine
  A_3125_KCU04 : FB 14;	// Mon1: DigInpCont
  A_3125_MXZ01_SM : FB 14;	// Mon2: DigInpCont
  Mon3 : FB 14;	// spare
  Mon4 : FB 14;	// spare
  Mon5 : FB 14;	// spare
  Mon6 : FB 14;	// spare
  A_3125_MXZ01 : FB 12;	// Motor: Motor
END_VAR
BEGIN
NETWORK
TITLE = Call SSW
      UC    "GCS7_M_Motor6Mon";
END_FUNCTION_BLOCK

FUNCTION_BLOCK "A_3126_MXZ01MA_Code"	// FB 1019
TITLE = A_3126_MXZ01MA FAN 2
//COPYRIGHT:     (C) 2009  BUHLER AG, CH-9240 UZWIL, SWITZERLAND
//
//PRODUCT:       WinCoS_BIW01_09
//
//TITLE:         FAN 2
// 
//--------------------------------------------------------------------------------
// 
//IDENT:         AUTHOR:             DEPT:                             DATE:
// 
//P01_FB1019.1.0 K.Renz              CSB41                             07.Okt.2009
//               1st Release
// 
//--------------------------------------------------------------------------------
// 
//PURPOSE: 
// 
//MANUAL : 
// 
//RESTRICTIONS: 
// 
//--------------------------------------------------------------------------------
//
AUTHOR : KR
FAMILY : USW
VERSION : 0.0
VAR
  Ma : UDT 20500;	// Machine
  A_3126_KCU04 : FB 14;	// Mon1: DigInpCont
  A_3126_MXZ01_SM : FB 14;	// Mon2: DigInpCont
  Mon3 : FB 14;	// spare
  Mon4 : FB 14;	// spare
  Mon5 : FB 14;	// spare
  Mon6 : FB 14;	// spare
  A_3126_MXZ01 : FB 12;	// Motor: Motor
END_VAR
BEGIN
NETWORK
TITLE = Call SSW
      UC    "GCS7_M_Motor6Mon";
END_FUNCTION_BLOCK

FUNCTION_BLOCK "A_3225_MXZ01MA_Code"	// FB 1032
TITLE = A_3225_MXZ01MA FAN 1
//COPYRIGHT:     (C) 2009  BUHLER AG, CH-9240 UZWIL, SWITZERLAND
//
//PRODUCT:       WinCoS_BIW01_09
//
//TITLE:         FAN 1
// 
//--------------------------------------------------------------------------------
// 
//IDENT:         AUTHOR:             DEPT:                             DATE:
// 
//P01_FB1032.1.0 K.Renz              CSB41                             06.Nov.2009
//               1st Release
// 
//--------------------------------------------------------------------------------
// 
//PURPOSE: 
// 
//MANUAL : 
// 
//RESTRICTIONS: 
// 
//--------------------------------------------------------------------------------
//
AUTHOR : KR
FAMILY : USW
VERSION : 0.0
VAR
  Ma : UDT 20500;	// Machine
  A_3225_KCU04 : FB 14;	// Mon1: DigInpCont
  A_3225_MXZ01_SM : FB 14;	// Mon2: DigInpCont
  Mon3 : FB 14;	// spare
  Mon4 : FB 14;	// spare
  Mon5 : FB 14;	// spare
  Mon6 : FB 14;	// spare
  A_3225_MXZ01 : FB 12;	// Motor: Motor
END_VAR
BEGIN
NETWORK
TITLE = Call SSW
      UC    "GCS7_M_Motor6Mon";
END_FUNCTION_BLOCK

FUNCTION_BLOCK "A_3226_MXZ01MA_Code"	// FB 1033
TITLE = A_3226_MXZ01MA FAN 2
//COPYRIGHT:     (C) 2009  BUHLER AG, CH-9240 UZWIL, SWITZERLAND
//
//PRODUCT:       WinCoS_BIW01_09
//
//TITLE:         FAN 2
// 
//--------------------------------------------------------------------------------
// 
//IDENT:         AUTHOR:             DEPT:                             DATE:
// 
//P01_FB1033.1.0 K.Renz              CSB41                             06.Nov.2009
//               1st Release
// 
//--------------------------------------------------------------------------------
// 
//PURPOSE: 
// 
//MANUAL : 
// 
//RESTRICTIONS: 
// 
//--------------------------------------------------------------------------------
//
AUTHOR : KR
FAMILY : USW
VERSION : 0.0
VAR
  Ma : UDT 20500;	// Machine
  A_3226_KCU04 : FB 14;	// Mon1: DigInpCont
  A_3226_MXZ01_SM : FB 14;	// Mon2: DigInpCont
  Mon3 : FB 14;	// spare
  Mon4 : FB 14;	// spare
  Mon5 : FB 14;	// spare
  Mon6 : FB 14;	// spare
  A_3226_MXZ01 : FB 12;	// Motor: Motor
END_VAR
BEGIN
NETWORK
TITLE = Call SSW
      UC    "GCS7_M_Motor6Mon";
END_FUNCTION_BLOCK

DATA_BLOCK DB 52
TITLE = PLC: System informations
//COPYRIGHT:    (C) 2000 BY  BUHLER AG
//                           CH-9240 UZWIL  SWITZERLAND
//
//PRODUCT:      STD_MU664
//
//TITLE:        PLC: System informations
//
//              PLC: Systeminformationen
//
//
//--------------------------------------------------------------------------------
//
//IDENT:        AUTHOR:             DEPT:                              DATE:
//
//STD_DB050.1.1 Ph. Engler          MU664                              21-Dec-2000
//              ColdStart signals and counter integrated
//STD_DB050.1A  Ph. Engler          MU664                              05-Jan-2000
//              1st Release
//
//--------------------------------------------------------------------------------
//
//PURPOSE:  
//MANUAL : 
//CODE   :
//RESTRICTIONS:
//
//--------------------------------------------------------------------------------
//
//
//
//
//
//
//
AUTHOR : PE
FAMILY : GEN
NAME : SystemDB
VERSION : 9.9
  STRUCT
   Spare00 : WORD ;
   Startup : STRUCT
    CmdNewstartMan : BOOL ;	//Manual newstart active
    CmdNewstartAuto : BOOL ;	//Automatic newstart active
    CmdRestartMan : BOOL ;	//Manual restart requested
    CmdRestartAuto : BOOL ;	//Automatic restart requested
    CmdColdstartMan : BOOL ;	//Manual coldstart requested
    CmdColdstartAuto : BOOL ;	//Automatic coldstart requested
    NotUsed06 : BOOL ;
    NotUsed07 : BOOL ;
    CmdStartTestMode : BOOL ;	//Starts the test mode
   END_STRUCT ;
   StartupCounter : STRUCT
    NewstartMan : INT ;	//Number of manual newstart startups
    NewstartAuto : INT ;	//Number of automatic newstart startups
    RestartMan : INT ;	//Number of manual restart startups
    RestartAuto : INT ;	//Number of automatic restart startups
    ColdstartMan : INT ;	//Number of manual coldstart startups
    ColdstartAuto : INT ;	//Number of automatic coldstart startups
    NotUsed07 : INT ;
    NotUsed08 : INT ;
    NotUsed09 : INT ;
    NotUsed10 : INT ;
    NotUsed11 : INT ;
    NotUsed12 : INT ;
   END_STRUCT ;
   Hardware : STRUCT
    PLCBatteryFailure : BOOL ;
    NotUsed09 : BOOL ;
    NotUsed10 : BOOL ;
    NotUsed11 : BOOL ;
    NotUsed12 : BOOL ;
    NotUsed13 : BOOL ;
    NotUsed14 : BOOL ;
    NotUsed15 : BOOL ;
    VoltageOk : BOOL ;	//Control voltage ok
    EsGeneralOk : BOOL ;	//General emergency stop ok
    PowerOk : BOOL ;	//Power supply motor contactor panels ok
    FuseOk : BOOL ;	//Mini circuit breakers ok
    PlcOk : BOOL ;	//PLC ok
    FireOk : BOOL ;	//No fire alarms
    SmokeOk : BOOL ;	//No smoke alarms
    ExflapsOk : BOOL ;	//Explosion flaps ok
   END_STRUCT ;
   HardwareStop : STRUCT
    UnloadingSteeping : BOOL ;	//Stop from Hardware circuit cabinet +C19
    UnloadingGeminating : BOOL ;	//Stop from Hardware circuit cabinet +C29
    NotUsed02 : BOOL ;
    NotUsed03 : BOOL ;
    NotUsed04 : BOOL ;
    NotUsed05 : BOOL ;
    NotUsed06 : BOOL ;
    NotUsed07 : BOOL ;
    General : BOOL ;	//Stop from Hardware all circuits
    General_C1 : BOOL ;	//Stop from Hardware circuit cabinet +C1
    Steeping : BOOL ;	//Stop from Hardware circuit cabinet +C11
    Germinating_1 : BOOL ;	//Stop from Hardware circuit cabinet +C21
    Germinating_2 : BOOL ;	//Stop from Hardware circuit cabinet +C22
    Germinating_3 : BOOL ;	//Stop from Hardware circuit cabinet +C23
    Germinating_4 : BOOL ;	//Stop from Hardware circuit cabinet +C24
    Germinating_5 : BOOL ;	//Stop from Hardware circuit cabinet +C25
   END_STRUCT ;
   GlobalFlags : STRUCT
    Germinating_6 : BOOL ;	//Stop from Hardware circuit cabinet +C26
    Germinating_7 : BOOL ;	//Stop from Hardware circuit cabinet +C27
    Germinating_8 : BOOL ;	//Stop from Hardware circuit cabinet +C28
    Kilning_1 : BOOL ;	//Stop from Hardware circuit cabinet +C31
    Kilning_2 : BOOL ;	//Stop from Hardware circuit cabinet +C32
    UnloadingKilning : BOOL ;	//Stop from Hardware circuit cabinet +C39
    NotUsed14 : BOOL ;
    DEC1_EXP1 : BOOL ;	//Stop from Hardware circuit cabinet +C41
    StaTest : BOOL ;	//Activates the test mode
    StaLOGOff : BOOL ;
    NotUsed02 : BOOL ;
    NotUsed03 : BOOL ;
    NotUsed04 : BOOL ;
    NotUsed05 : BOOL ;
    NotUsed06 : BOOL ;
    StaProtocolling : BOOL ;	//Activates the protocolling functionality of the elements
   END_STRUCT ;
   TestFunctions : STRUCT
    StaPLC1ComSimulation : BOOL ;
    StaPLC2ComSimulation : BOOL ;
    StaPLC3ComSimulation : BOOL ;
    StaPLC4ComSimulation : BOOL ;
    StaPLC5ComSimulation : BOOL ;
    StaPLC6ComSimulation : BOOL ;
    StaPLC7ComSimulation : BOOL ;
    StaPLC8ComSimulation : BOOL ;
    StaIOManager : BOOL ;	//IO's simulated with the IO-Manager
    StaHardware : BOOL ;	//IO's connected to the real hardware
    StaCWASimulation : BOOL ;	//CWA-Simulator on
    StaIOSimuli : BOOL ;	//IO's simulated with the IOSimuli
    StaDPSimulation : BOOL ;	//Simulation of DP-Scales
    StaWinAC : BOOL ;	//Testing on a WinAC
    NotUsed06 : BOOL ;
    StaPCDirectInhouseTest : BOOL ;	//Direct control channel for inhouse test
    StaPLC9ComSimulation : BOOL ;
    StaPLC10ComSimulation : BOOL ;
    StaPLC11ComSimulation : BOOL ;
    StaPLC12ComSimulation : BOOL ;
    StaPLC13ComSimulation : BOOL ;
    StaPLC14ComSimulation : BOOL ;
    StaPLC15ComSimulation : BOOL ;
    StaPLC16ComSimulation : BOOL ;
   END_STRUCT ;
   PlantID : STRUCT
    Product : ARRAY  [1 .. 15 ] OF //i.e. MELE_SMU01_99
    CHAR ;
    PlcNr : INT  := 1;
    GCSRelease : INT  := 2;
   END_STRUCT ;
  END_STRUCT ;	
BEGIN
   PlantID.Product[1] := 'M';
   PlantID.Product[2] := 'E';
   PlantID.Product[3] := 'L';
   PlantID.Product[4] := 'E';
   PlantID.Product[5] := '_';
   PlantID.Product[6] := 'S';
   PlantID.Product[7] := 'M';
   PlantID.Product[8] := 'U';
   PlantID.Product[9] := '0';
   PlantID.Product[10] := '1';
   PlantID.Product[11] := '_';
   PlantID.Product[12] := '9';
   PlantID.Product[13] := '9';
   PlantID.Product[14] := ' ';
   PlantID.Product[15] := ' ';
   PlantID.PlcNr := 1;
   PlantID.GCSRelease := 2;
END_DATA_BLOCK

DATA_BLOCK "G270M"	// DB 370
TITLE = DBG270M  AIR SHUT SLIDE KILN 1
//COPYRIGHT:    (C) 2009  BUHLER AG, CH-9240 UZWIL, SWITZERLAND
//
//PRODUCT:      WinCoS_BIW01_09
//
//TITLE:        AIR SHUT SLIDE KILN 1
//                Machine group DB
//                Maschinengruppen-DB
//
//-------------------------------------------------------------------------
//
//IDENT:        AUTHOR:             DEPT:             DATE:
//
//P01_DB370.1.0 K.Renz              CSB41             06.Okt.2009
//              1st Release
//
//-------------------------------------------------------------------------
//
//PURPOSE: 
//
//MANUAL : 
//
//RESTRICTIONS: 
//
//-------------------------------------------------------------------------
//
AUTHOR : KR
FAMILY : USW
NAME : DBG270M
VERSION : 0.0
"G270M_Code"
BEGIN
END_DATA_BLOCK

DATA_BLOCK "G271M"	// DB 371
TITLE = DBG271M  FAN KILN 1
//COPYRIGHT:    (C) 2009  BUHLER AG, CH-9240 UZWIL, SWITZERLAND
//
//PRODUCT:      WinCoS_BIW01_09
//
//TITLE:        FAN KILN 1
//                Machine group DB
//                Maschinengruppen-DB
//
//-------------------------------------------------------------------------
//
//IDENT:        AUTHOR:             DEPT:             DATE:
//
//P01_DB371.1.0 K.Renz              CSB41             09.Apr.2010
//              1st Release
//
//-------------------------------------------------------------------------
//
//PURPOSE: 
//
//MANUAL : 
//
//RESTRICTIONS: 
//
//-------------------------------------------------------------------------
//
AUTHOR : KR
FAMILY : USW
NAME : DBG271M
VERSION : 0.0
"G271M_Code"
BEGIN
END_DATA_BLOCK

DATA_BLOCK "G297M"	// DB 397
TITLE = DBG297M  FAN KILN 2
//COPYRIGHT:    (C) 2009  BUHLER AG, CH-9240 UZWIL, SWITZERLAND
//
//PRODUCT:      WinCoS_BIW01_09
//
//TITLE:        FAN KILN 2
//                Machine group DB
//                Maschinengruppen-DB
//
//-------------------------------------------------------------------------
//
//IDENT:        AUTHOR:             DEPT:             DATE:
//
//P01_DB397.1.0 K.Renz              CSB41             09.Apr.2010
//              1st Release
//
//-------------------------------------------------------------------------
//
//PURPOSE: 
//
//MANUAL : 
//
//RESTRICTIONS: 
//
//-------------------------------------------------------------------------
//
AUTHOR : KR
FAMILY : USW
NAME : DBG297M
VERSION : 0.0
"G297M_Code"
BEGIN
END_DATA_BLOCK

ORGANIZATION_BLOCK OB 1
TITLE = "Main Program Sweep (Cycle)"
VERSION : 0.1
VAR_TEMP
  OB1_EV_CLASS : BYTE ;	//Bits 0-3 = 1 (Coming event), Bits 4-7 = 1 (Event class 1)
  OB1_SCAN_1 : BYTE ;	//1 (Cold restart scan 1 of OB 1), 3 (Scan 2-n of OB 1)
  OB1_PRIORITY : BYTE ;	//Priority of OB Execution
  OB1_OB_NUMBR : BYTE ;	//1 (Organization block 1, OB1)
  OB1_RESERVED_1 : BYTE ;	//Reserved for system
  OB1_RESERVED_2 : BYTE ;	//Reserved for system
  OB1_PREV_CYCLE : INT ;	//Cycle time of previous OB1 scan (milliseconds)
  OB1_MIN_CYCLE : INT ;	//Minimum cycle time of OB1 (milliseconds)
  OB1_MAX_CYCLE : INT ;	//Maximum cycle time of OB1 (milliseconds)
  OB1_DATE_TIME : DATE_AND_TIME ;	//Date and time OB1 started
END_VAR
BEGIN
// (block stored without names or comments; labels and parameter names are numbered)
END_ORGANIZATION_BLOCK

SYMBOL_TABLE
"G003G"	DB 103	FB 103	// Group-DB  PLC monitoring
"G269M"	DB 369	FB 369	// Group-DB  TEMPERATURE MES. KILN 1
"G285M"	DB 385	FB 385	// Group-DB  MAIN ASPIRATION 6181 - DEC1
"G003G_Code"	FB 103	FB 103	// Group-FB  PLC monitoring
"G269M_Code"	FB 369	FB 369	// Group-FB  TEMPERATURE MES. KILN 1
"G285M_Code"	FB 385	FB 385	// Group-FB  MAIN ASPIRATION 6181 - DEC1
END_SYMBOL_TABLE

FUNCTION_BLOCK "G003G_Code"	// FB 103
TITLE = G003G PLC monitoring
//COPYRIGHT:    (C) 2009  BUHLER AG, CH-9240 UZWIL, SWITZERLAND
//
//PRODUCT:      WinCoS_BIW01_09
//
//TITLE:        PLC monitoring
//                General group control
//                Allgemeine Gruppensteuerung
// 
//--------------------------------------------------------------------------------
// 
//IDENT:        AUTHOR:             DEPT:                              DATE:
// 
//P01_FB103.1.0 K.Renz              CSB41                              29.Sep.2009
//             1st Release
// 
//--------------------------------------------------------------------------------
// 
//PURPOSE: 
// 
//MANUAL : 
// 
//RESTRICTIONS: 
// 
//--------------------------------------------------------------------------------
//
AUTHOR : KR
FAMILY : USW
VERSION : 9.9
VAR
  Gr : FB 10;	//Standard interface to group
  InOutValue1 : DINT ;	//Data for user
  InOutValue2 : DINT ;	//Data for user
  OutWayConflict : BOOL ;	//Data for user
  OutSelectionOk : BOOL ;	//Data for user
  CmdNewValue : BOOL ;	//Data for user
  CmdNewJob : BOOL ;	//Data for user
  OutCodeOK : BOOL ;	//Data for user
  InEndOfJob : BOOL ;	//Data for user
  staWayOk : BOOL ;	//Data for user
  EdgeStartRelease : BOOL ;	//Data for user
  USW8 : BOOL ;	//Data for user
  USW9 : BOOL ;	//Data for user
  USW10 : BOOL ;	//Data for user
  USW11 : BOOL ;	//Data for user
  USW12 : BOOL ;	//Data for user
  USW13 : BOOL ;	//Data for user
  USW14 : BOOL ;	//Data for user
  USW15 : BOOL ;	//Data for user
  G_PLC : FB 14;	// DigInpCont
  G_PS_BAT : FB 14;	// DigInpCont
END_VAR
VAR_TEMP
  tmpEnable : BOOL ;
  tmpFlag : BOOL ;
  tmpCmdNext : BOOL ;
  tmpLocal : BOOL ;
  tmpAspOk : BOOL ;
  tmpHWStop : BOOL ;
  tmpInstanzDBNo : INT ;
END_VAR
BEGIN
NETWORK
TITLE =
NETWORK
TITLE = Read command from group control
//Parameter
      SET;
      R     DB9.DBX 50.2;
      R     DB9.DBX 90.2;
      S     DB9.DBX 130.2;
      R     DB9.DBX 10.2;
      S     DB9.DBX 170.2;
      R     DIX [AR2,P#32.0];
      R     DIX [AR2,P#32.1];
      S     DIX [AR2,P#32.2];
//Command
      A     DB9.DBX 290.2;
      =     DIX [AR2,P#14.0];
      A     DB9.DBX 250.2;
      =     DIX [AR2,P#15.4];
      A     DB9.DBX 370.2;
      R     DB9.DBX 370.2;
      S     DIX [AR2,P#15.3];
      A     DB9.DBX 330.2;
      R     DB9.DBX 330.2;
      S     DIX [AR2,P#15.2];
      A     DB9.DBX 410.2;
      O     DB9.DBX 250.2;
      R     DB9.DBX 410.2;
      S     DIX [AR2,P#14.7];
      A     DB9.DBX 730.2;
      R     DB9.DBX 730.2;
      S     DIX [AR2,P#14.1];
//Init Line Number
      A     DB9.DBX 170.2;
      JCN   WE00;
      L     0;
      T     DIW [AR2,P#24.0];
WE00: NOP   0;
NETWORK
TITLE = Call Methode Control
// 1. Handle Interface PCControl      
// 2. Prepare mode --> ModePassive,ModeActive,ModeIdling      
// 3. Reset global flags of the group
      BLD   14;
      =     L 10.0;
      L     DINO;
      T     LW 8;
      CDB;
      OPN   DI [LW 8];
      TAR2  LD 4;
      L     1;
      T     DIW [AR2,P#0.0];
      +AR2  P#0.0;
      UC    FB 10;
      LAR2  LD 4;
      CDB;
      BLD   15;
NETWORK
TITLE = Restart Idling Time
      CLR;
      S     DIX [AR2,P#14.2];
NETWORK
TITLE = Prepare global flags
NETWORK
TITLE = Set Pattern (Target position)
NETWORK
TITLE = Interlocking WayOk
NETWORK
TITLE = Interlocking Autostart
      CLR;
      R     DIX [AR2,P#18.4];
NETWORK
TITLE = Interlocking Enable
      A     DIX [AR2,P#14.0];
      =     DIX [AR2,P#18.0];
NETWORK
TITLE = Interlocking Next
      A     DIX [AR2,P#15.2];
      A     DIX [AR2,P#18.4];
      AN    DIX [AR2,P#19.6];
      =     #tmpCmdNext;
NETWORK
TITLE = Interlocking Local / HWStop
      A     DB50.DBX 31.2;
      =     #tmpHWStop;
      A     DIX [AR2,P#16.0];
      =     #tmpLocal;
NETWORK
TITLE = G_PLC : PLC System
      NOP   0;
//-InLocal---
      A     #tmpLocal;
      =     DIX [AR2,P#63.4];
// 
//-Monitoring---
      SET;
      =     DIX [AR2,P#62.0];
// 
//-PreAlarm---
//  CLR
//  =      #G_PLC.InPreAlarmTrue 
// 
//-Additional commands---
//      CLR
//      S     #G_PLC.CmdRunTimeOutTime
// 
//-Read inputs---
      SET;
      =     DIX [AR2,P#62.6];
// 
//-Set Parameters---
// 
//-Call object control---
      BLD   14;
// 
//-Write outputs---
      =     L 10.0;
      L     DINO;
      T     LW 8;
      CDB;
      OPN   DI [LW 8];
      TAR2  LD 4;
      +AR2  P#60.0;
      UC    FB 14;
      LAR2  LD 4;
      CDB;
      BLD   15;
NETWORK
TITLE = G_PS_BAT : PLC Powersupply battery monitoring
      NOP   0;
//-InLocal---
      A     #tmpLocal;
      =     DIX [AR2,P#97.4];
// 
//-Monitoring---
      SET;
      =     DIX [AR2,P#96.0];
// 
//-PreAlarm---
//  CLR
//  =      #G_PS_BAT.InPreAlarmTrue 
// 
//-Additional commands---
//      CLR
//      S     #G_PS_BAT.CmdRunTimeOutTime
// 
//-Read inputs---
      AN    DB50.DBX 28.0;
      =     DIX [AR2,P#96.6];
// 
//-Set Parameters---
// 
//-Call object control---
      BLD   14;
// 
//-Write outputs---
      =     L 10.0;
      L     DINO;
      T     LW 8;
      CDB;
      OPN   DI [LW 8];
      TAR2  LD 4;
      +AR2  P#94.0;
      UC    FB 14;
      LAR2  LD 4;
      CDB;
      BLD   15;
NETWORK
TITLE = Test Fault
      A     DIX [AR2,P#65.4];
      =     DIX [AR2,P#19.2];
NETWORK
TITLE = Test Warning
      A     DIX [AR2,P#65.0];
      O     DIX [AR2,P#99.4];
      O     DIX [AR2,P#99.0];
      =     DIX [AR2,P#17.6];
NETWORK
TITLE = Test Stopped
      SET;
      =     DIX [AR2,P#19.0];
NETWORK
TITLE = Test Started
      A(;
      O     DIX [AR2,P#65.2];
      O     DIX [AR2,P#65.3];
      );
      A(;
      O     DIX [AR2,P#99.2];
      O     DIX [AR2,P#99.3];
      );
      AN    DIX [AR2,P#19.2];
      =     DIX [AR2,P#19.1];
NETWORK
TITLE = Enable Previous Group
      A     DIX [AR2,P#19.1];
      =     DIX [AR2,P#18.7];
NETWORK
TITLE = Call Methode State
//1. Make State of the group: This function use the signals:
//        Gr.VarStopped, Gr.VarStarted, Gr.VarFault
//2.Reset Commands to group: e.g.CmdFaultReset
      BLD   14;
      =     L 10.0;
      L     DINO;
      T     LW 8;
      CDB;
      OPN   DI [LW 8];
      TAR2  LD 4;
      L     2;
      T     DIW [AR2,P#0.0];
      +AR2  P#0.0;
      UC    FB 10;
      LAR2  LD 4;
      CDB;
      BLD   15;
NETWORK
TITLE = Init
      SET;
      R     DIX [AR2,P#58.2];
      R     DIX [AR2,P#58.3];
NETWORK
TITLE = Write data to group control
      A     DIX [AR2,P#17.0];
      =     DB9.DBX 450.2;
      A     DIX [AR2,P#17.2];
      =     DB9.DBX 490.2;
      A     DIX [AR2,P#17.4];
      =     DB9.DBX 530.2;
      A     DIX [AR2,P#17.6];
      =     DB9.DBX 570.2;
      A     DIX [AR2,P#18.5];
      =     DB9.DBX 610.2;
      A     DIX [AR2,P#18.2];
      =     DB9.DBX 850.2;
      A     DIX [AR2,P#18.3];
      =     DB9.DBX 810.2;
      A     DIX [AR2,P#17.5];
      =     DB9.DBX 770.2;
      A     DIX [AR2,P#18.4];
      =     DB9.DBX 890.2;
      A     DIX [AR2,P#19.3];
      =     DB9.DBX 930.2;
NETWORK
TITLE = End of block
      BE;
END_FUNCTION_BLOCK

FUNCTION_BLOCK "G269M_Code"	// FB 369
TITLE = G269M TEMPERATURE MES. KILN 1
//COPYRIGHT:    (C) 2009  BUHLER AG, CH-9240 UZWIL, SWITZERLAND
//
//PRODUCT:      WinCoS_BIW01_09
//
//TITLE:        TEMPERATURE MES. KILN 1
//                Machine group control
//                Maschinengruppensteuerung
// 
//--------------------------------------------------------------------------------
// 
//IDENT:        AUTHOR:             DEPT:                              DATE:
// 
//P01_FB369.1.0 K.Renz              CSB41                              30.Sep.2009
//             1st Release
// 
//--------------------------------------------------------------------------------
// 
//PURPOSE: 
// 
//MANUAL : 
// 
//RESTRICTIONS: 
// 
//--------------------------------------------------------------------------------
//
AUTHOR : KR
FAMILY : USW
VERSION : 9.9
VAR
  Gr : FB 10;	//Standard interface to group
  InOutValue1 : DINT ;	//Data for user
  InOutValue2 : DINT ;	//Data for user
  OutWayConflict : BOOL ;	//Data for user
  OutSelectionOk : BOOL ;	//Data for user
  CmdNewValue : BOOL ;	//Data for user
  CmdNewJob : BOOL ;	//Data for user
  OutCodeOK : BOOL ;	//Data for user
  InEndOfJob : BOOL ;	//Data for user
  staWayOk : BOOL ;	//Data for user
  EdgeStartRelease : BOOL ;	//Data for user
  read_3191 : BOOL ;	//Data for user
  USW9 : BOOL ;	//Data for user
  USW10 : BOOL ;	//Data for user
  USW11 : BOOL ;	//Data for user
  USW12 : BOOL ;	//Data for user
  USW13 : BOOL ;	//Data for user
  USW14 : BOOL ;	//Data for user
  USW15 : BOOL ;	//Data for user
  A_3191_BTE01 : FB 19;	// AnaInp
  A_3191_BTE05 : FB 19;	// AnaInp
  A_3191_BTE07 : FB 19;	// AnaInp
  A_3191_BTE08 : FB 19;	// AnaInp
  A_3191_BTE10 : FB 19;	// AnaInp
  A_3191_BTE11 : FB 19;	// AnaInp
  A_3191_BTE12 : FB 19;	// AnaInp
  A_3191_BTE06 : FB 19;	// AnaInp
END_VAR
VAR_TEMP
  tmpEnable : BOOL ;
  tmpFlag : BOOL ;
  tmpCmdNext : BOOL ;
  tmpLocal : BOOL ;
  tmpAspOk : BOOL ;
  tmpHWStop : BOOL ;
  tmpInstanzDBNo : INT ;
END_VAR
BEGIN
NETWORK
TITLE =
NETWORK
TITLE = Read command from group control
//Parameter
      SET;
      S     DB9.DBX 83.4;
      R     DB9.DBX 123.4;
      R     DB9.DBX 163.4;
      R     DB9.DBX 43.4;
      R     DB9.DBX 203.4;
      S     DIX [AR2,P#32.0];
      R     DIX [AR2,P#32.1];
      R     DIX [AR2,P#32.2];
//Command
      A     DB9.DBX 323.4;
      =     DIX [AR2,P#14.0];
      A     DB9.DBX 283.4;
      =     DIX [AR2,P#15.4];
      A     DB9.DBX 403.4;
      R     DB9.DBX 403.4;
      S     DIX [AR2,P#15.3];
      A     DB9.DBX 363.4;
      R     DB9.DBX 363.4;
      S     DIX [AR2,P#15.2];
      A     DB9.DBX 443.4;
      O     DB9.DBX 283.4;
      R     DB9.DBX 443.4;
      S     DIX [AR2,P#14.7];
      A     DB9.DBX 763.4;
      R     DB9.DBX 763.4;
      S     DIX [AR2,P#14.1];
//Init Line Number
      A     DB9.DBX 203.4;
      JCN   WE00;
      L     0;
      T     DIW [AR2,P#24.0];
WE00: NOP   0;
NETWORK
TITLE = Call Methode Control
// 1. Handle Interface PCControl      
// 2. Prepare mode --> ModePassive,ModeActive,ModeIdling      
// 3. Reset global flags of the group
      BLD   14;
      =     L 10.0;
      L     DINO;
      T     LW 8;
      CDB;
      OPN   DI [LW 8];
      TAR2  LD 4;
      L     1;
      T     DIW [AR2,P#0.0];
      +AR2  P#0.0;
      UC    FB 10;
      LAR2  LD 4;
      CDB;
      BLD   15;
NETWORK
TITLE = Restart Idling Time
      L     DIW [AR2,P#36.0];
      L     2;
      >=I;
      JC    IdTm;
      T     DIW [AR2,P#36.0];
IdTm: NOP   0;
      CLR;
      S     DIX [AR2,P#14.2];
NETWORK
TITLE = Prepare global flags
NETWORK
TITLE = Set Pattern (Target position)
NETWORK
TITLE = Interlocking WayOk
NETWORK
TITLE = Interlocking Autostart
      CLR;
      R     DIX [AR2,P#18.4];
NETWORK
TITLE = Interlocking Enable
      A     DIX [AR2,P#14.0];
      =     DIX [AR2,P#18.0];
NETWORK
TITLE = Interlocking Next
      A     DIX [AR2,P#15.2];
      A     DIX [AR2,P#18.4];
      AN    DIX [AR2,P#19.6];
      =     #tmpCmdNext;
NETWORK
TITLE = Interlocking Local / HWStop
      A     DB50.DBX 32.3;
      =     #tmpHWStop;
      A     DIX [AR2,P#16.0];
      O     #tmpHWStop;
      =     #tmpLocal;
NETWORK
TITLE = =A-3191-BTE01 : AIR TEMPERATURE BELOW FLOOR
      NOP   0;
//-InLocal---
      A     #tmpLocal;
      =     DIX [AR2,P#63.4];
//-Monitoring--- 
      A     DB922.DBX 410.0;
      =     DIX [AR2,P#62.0];
      =     DIX [AR2,P#62.1];
      CLR;
      =     DIX [AR2,P#62.2];
      A     DB922.DBX 410.0;
      =     DIX [AR2,P#62.3];
      =     DIX [AR2,P#62.4];
//MW 2010.04.08
      SET;
      =     DIX [AR2,P#84.7];
      =     DIX [AR2,P#85.1];
      CLR;
      =     DIX [AR2,P#84.6];
      =     DIX [AR2,P#85.3];
      =     DIX [AR2,P#85.7];
      =     DIX [AR2,P#85.2];
// 
//-Read inputs---
      L     PIW 936;
      L     50;
      -I;
      T     DIW [AR2,P#66.0];
      A     DB50.DBX 32.3;
      =     DIX [AR2,P#63.0];
      A     DB51.DBX 11.3;
      =     DIX [AR2,P#63.1];
// 
//-Set Parameters---
      SET;	//BRT20100828 - kein Alarmhorn wenn Warning
      =     DB369.DBX 84.5;
      AN    DB922.DBX 410.0;
      JC    fui;
// Toleranzband -1,5°C Temperatur unter der Horde
      L     DB922.DBD 1700;
      L     L#10;
      *D;
      L     L#150;	// =1,5°C
      -D;
      T     DID [AR2,P#102.0];
// Toleranzband +1,5°C Temperatur unter der Horde
      L     DB922.DBD 1700;
      L     L#10;
      *D;
      L     L#150;	// =1,5°C
      +D;
      T     DID [AR2,P#106.0];
      JU    hui;
fui:  NOP   0;
      L     L#-10000;	// -100,00°C
      T     DID [AR2,P#98.0];
      L     L#0;	// 0,00°C
      T     DID [AR2,P#102.0];
      L     L#9900;	// 99,00°C
      T     DID [AR2,P#106.0];
      L     L#10000;	// 100,00°C
      T     DID [AR2,P#110.0];
hui:  NOP   0;
// 
//-Call object control---
      BLD   14;
// 
//-Write outputs---
// Schaltpunkt zu Oeffnen der Defrosterklappe
      =     L 10.0;
      L     DINO;	// =70,00°C
      T     LW 8;
      CDB;
      OPN   DI [LW 8];
      TAR2  LD 4;
      +AR2  P#60.0;
      UC    FB 19;
      LAR2  LD 4;
      CDB;
      BLD   15;
      L     DIW [AR2,P#68.0];
      L     7000;
      >=I;
      =     DB922.DBX 421.0;
NETWORK
TITLE = =A-3191-BTE05 : AIR TEMPERATURE DIFFUSOR FAN 1
      NOP   0;
//-InLocal---
      A     #tmpLocal;
      =     DIX [AR2,P#151.4];
//-Monitoring--- 
      CLR;
      =     DIX [AR2,P#150.0];
      CLR;
      =     DIX [AR2,P#150.1];
      CLR;
      =     DIX [AR2,P#150.2];
      CLR;
      =     DIX [AR2,P#150.3];
      A     DB922.DBX 410.0;
      =     DIX [AR2,P#150.4];
// 
//-Read inputs---
      L     PIW 938;
      L     50;
      -I;
      T     DIW [AR2,P#154.0];
      A     DB50.DBX 32.3;
      =     DIX [AR2,P#151.0];
      A     DB51.DBX 11.3;
      =     DIX [AR2,P#151.1];
// 
//-Set Parameters---
      A     DB922.DBX 410.0;
      R     DIX [AR2,P#172.5];
      AN    DB922.DBX 410.0;
      ON    DB371.DBX 417.2;
      ON    DB376.DBX 341.2;
      JC    fui1;
// Toleranzband -3,5°C Temperatur unter der Horde
      L     DB922.DBD 1700;
      L     L#10;
      *D;
      L     L#350;	// =3,5°C
      -D;
      T     DID [AR2,P#190.0];
// Toleranzband +3,5°C Temperatur unter der Horde
      L     DB922.DBD 1700;
      L     L#10;
      *D;
      L     L#350;	// =3,5°C
      +D;
      T     DID [AR2,P#194.0];
      JU    hui1;
fui1: NOP   0;
      L     L#-10000;	// -100,00°C
      T     DID [AR2,P#186.0];
      L     L#0;	// 0,00°C
      T     DID [AR2,P#190.0];
      L     L#9900;	// 99,00°C
      T     DID [AR2,P#194.0];
      L     L#10000;	// 100,00°C
      T     DID [AR2,P#198.0];
hui1: NOP   0;
// 
//-Call object control---
      BLD   14;
// 
//-Write outputs---
      =     L 10.0;
      L     DINO;
      T     LW 8;
      CDB;
      OPN   DI [LW 8];
      TAR2  LD 4;
      +AR2  P#148.0;
      UC    FB 19;
      LAR2  LD 4;
      CDB;
      BLD   15;
NETWORK
TITLE = =A-3191-BTE07 : AIR TEMPERATURE ABOVE FLOOR
      NOP   0;
//-InLocal---
      A     #tmpLocal;
      =     DIX [AR2,P#239.4];
//-Monitoring--- 
      CLR;
      =     DIX [AR2,P#238.0];
      CLR;
      =     DIX [AR2,P#238.1];
      CLR;
      =     DIX [AR2,P#238.2];
      A     DB922.DBX 410.0;
      =     DIX [AR2,P#238.3];
      A     DB922.DBX 410.0;
      AN    DIX [AR2,P#240.4];
      =     DIX [AR2,P#261.1];
      A     DB922.DBX 410.0;
      =     DIX [AR2,P#238.4];
      =     DIX [AR2,P#261.7];
      A     DB922.DBX 410.0;
      AN    DIX [AR2,P#240.4];
      =     DIX [AR2,P#261.2];
// 
//-Read inputs---
      L     PIW 940;
      T     DIW [AR2,P#242.0];
      A     DB50.DBX 32.3;
      =     DIX [AR2,P#239.0];
      A     DB51.DBX 11.3;
      =     DIX [AR2,P#239.1];
// 
//-Set Parameters---
      A     DB922.DBX 410.0;
      R     DIX [AR2,P#260.5];
      AN    DB922.DBX 410.0;
      JC    psp;
//      L     "MAL1S032Par".RecipeHeader.WarningTempAboveFloor
      L     L#900;	// 90,00°C
      L     L#10;
      *D;
      T     DID [AR2,P#282.0];
      L     DID [AR2,P#282.0];
      L     L#500;
      +D;
      T     DID [AR2,P#286.0];
psp:  NOP   0;
      A     DB922.DBX 410.0;
      JC    npsp;
      L     L#-10000;	// -100,00°C
      T     DID [AR2,P#274.0];
      L     L#0;	// 0,00°C
      T     DID [AR2,P#278.0];
      L     L#9900;	// 99,00°C
      T     DID [AR2,P#282.0];
      L     L#10000;	// 100,00°C
      T     DID [AR2,P#286.0];
npsp: NOP   0;
// 
//-Call object control---
      BLD   14;
// 
//-Write outputs---
      =     L 10.0;
      L     DINO;
      T     LW 8;
      CDB;
      OPN   DI [LW 8];
      TAR2  LD 4;
      +AR2  P#236.0;
      UC    FB 19;
      LAR2  LD 4;
      CDB;
      BLD   15;
NETWORK
TITLE = =A-3191-BTE08 : AIR TEMPERATURE AFTER BURNER 1
//      NOP   0
////-InLocal---
//      U     #tmpLocal
//      =     #A_3191_BTE08.InLocal
//
////-Monitoring--- 
//      CLR   
//      =     #A_3191_BTE08.InMonLL
//      CLR   
//      =     #A_3191_BTE08.InMonL
//      CLR   
//      =     #A_3191_BTE08.InMonMid
//      CLR   
//      =     #A_3191_BTE08.InMonH
//      U     "MAL1S032Par".Par.FlagProcess.ProcessActive
//      =     #A_3191_BTE08.InMonHH
//// 
////-Read inputs---
//      L     "A_3191_BTE08_AI1"
//      T     #A_3191_BTE08.InpValue
//      U     "PLC_SystemDB".GlobalFlags.Kilning_1
//      =     #A_3191_BTE08.InHWStop
//      U     "PLC_DPInfo".Master[1].SlavesError[92]
//      =     #A_3191_BTE08.InDPFault
//// 
////-Set Parameters---
//      L     L#-10000                    // -100,00°C
//      T     #A_3191_BTE08.Par.ParLimitLL
//      L     L#0                         // 0,00°C
//      T     #A_3191_BTE08.Par.ParLimitL
//      L     L#9900                      // 99,00°C
//      T     #A_3191_BTE08.Par.ParLimitH
//      L     L#10000                     // 100,00°C
//      T     #A_3191_BTE08.Par.ParLimitHH
//// 
////-Call object control---
//      CALL  #A_3191_BTE08
//// 
////-Write outputs---
//
NETWORK
TITLE = =A-3191-BTE10 : AIR TEMPERATURE BEFORE BURNER 2
      NOP   0;
//-InLocal---
      A     #tmpLocal;
      =     DIX [AR2,P#415.4];
//-Monitoring--- 
      CLR;
      =     DIX [AR2,P#414.0];
      CLR;
      =     DIX [AR2,P#414.1];
      CLR;
      =     DIX [AR2,P#414.2];
      CLR;
      =     DIX [AR2,P#414.3];
      A     DB922.DBX 410.0;
      =     DIX [AR2,P#414.4];
// 
//-Read inputs---
      L     PIW 944;
      T     DIW [AR2,P#418.0];
      A     DB50.DBX 32.3;
      =     DIX [AR2,P#415.0];
      A     DB51.DBX 11.3;
      =     DIX [AR2,P#415.1];
// 
//-Set Parameters---
      L     L#-10000;	// -100,00°C
      T     DID [AR2,P#450.0];
      L     L#0;	// 0,00°C
      T     DID [AR2,P#454.0];
      L     L#9900;	// 99,00°C
      T     DID [AR2,P#458.0];
      L     L#10000;	// 100,00°C
      T     DID [AR2,P#462.0];
// 
//-Call object control---
      BLD   14;
// 
//-Write outputs---
      =     L 10.0;
      L     DINO;
      T     LW 8;
      CDB;
      OPN   DI [LW 8];
      TAR2  LD 4;
      +AR2  P#412.0;
      UC    FB 19;
      LAR2  LD 4;
      CDB;
      BLD   15;
NETWORK
TITLE = =A-3191-BTE11 : AIR TEMPERATURE AMBIENT AIR
      NOP   0;
//-InLocal---
      A     #tmpLocal;
      =     DIX [AR2,P#503.4];
//-Monitoring--- 
      SET;
      =     DIX [AR2,P#502.0];
      CLR;
      =     DIX [AR2,P#502.1];
      CLR;
      =     DIX [AR2,P#502.2];
      CLR;
      =     DIX [AR2,P#502.3];
      SET;
      =     DIX [AR2,P#502.4];
// 
//-Read inputs---
      L     PIW 946;
      T     DIW [AR2,P#506.0];
      A     DB50.DBX 32.3;
      =     DIX [AR2,P#503.0];
      A     DB51.DBX 11.3;
      =     DIX [AR2,P#503.1];
// 
//-Set Parameters---
      A     DB922.DBX 410.0;
      R     DIX [AR2,P#524.5];
      L     L#-10000;	// -100,00°C
      T     DID [AR2,P#538.0];
      L     L#0;	// 0,00°C
      T     DID [AR2,P#542.0];
      L     L#3200;	// 32,00°C
//      L     "MAL1Par".Values1.Value03   // Line Parameter --> not used!!
//      L     L#100
//      *D    
      T     DID [AR2,P#546.0];
      L     L#10000;	// 100,00°C
      T     DID [AR2,P#550.0];
// 
//-Call object control---
      BLD   14;
// 
//-Write outputs---
      =     L 10.0;
      L     DINO;
      T     LW 8;
      CDB;
      OPN   DI [LW 8];
      TAR2  LD 4;
      +AR2  P#500.0;
      UC    FB 19;
      LAR2  LD 4;
      CDB;
      BLD   15;
NETWORK
TITLE = =A-3191-BTE12 : AIR TEMPERATURE AFTER HEAT EXCHANGER FLAP
      NOP   0;
//-InLocal---
      A     #tmpLocal;
      =     DIX [AR2,P#591.4];
//-Monitoring--- 
      CLR;
      =     DIX [AR2,P#590.0];
      CLR;
      =     DIX [AR2,P#590.1];
      CLR;
      =     DIX [AR2,P#590.2];
      CLR;
      =     DIX [AR2,P#590.3];
      A     DB922.DBX 410.0;
      =     DIX [AR2,P#590.4];
// 
//-Read inputs---
      L     PIW 948;
      T     DIW [AR2,P#594.0];
      A     DB50.DBX 32.3;
      =     DIX [AR2,P#591.0];
      A     DB51.DBX 11.3;
      =     DIX [AR2,P#591.1];
// 
//-Set Parameters---
      L     L#-10000;	// -100,00°C
      T     DID [AR2,P#626.0];
      L     L#0;	// 0,00°C
      T     DID [AR2,P#630.0];
      L     L#9900;	// 99,00°C
      T     DID [AR2,P#634.0];
      L     L#10000;	// 100,00°C
      T     DID [AR2,P#638.0];
// 
//-Call object control---
      BLD   14;
// 
//-Write outputs---
      =     L 10.0;
      L     DINO;
      T     LW 8;
      CDB;
      OPN   DI [LW 8];
      TAR2  LD 4;
      +AR2  P#588.0;
      UC    FB 19;
      LAR2  LD 4;
      CDB;
      BLD   15;
NETWORK
TITLE = =A-3191-BTE06 : AIR TEMPERATURE DIFFUSOR FAN 2
      NOP   0;
//-InLocal---
      A     #tmpLocal;
      =     DIX [AR2,P#679.4];
//-Monitoring--- 
      CLR;
      =     DIX [AR2,P#678.0];
      CLR;
      =     DIX [AR2,P#678.1];
      CLR;
      =     DIX [AR2,P#678.2];
      CLR;
      =     DIX [AR2,P#678.3];
      A     DB922.DBX 410.0;
      =     DIX [AR2,P#678.4];
// 
//-Read inputs---
      L     PIW 950;
      L     50;
      -I;
      T     DIW [AR2,P#682.0];
      A     DB50.DBX 32.3;
      =     DIX [AR2,P#679.0];
      A     DB51.DBX 11.3;
      =     DIX [AR2,P#679.1];
// 
//-Set Parameters---
      A     DB922.DBX 410.0;
      R     DIX [AR2,P#700.5];
      AN    DB922.DBX 410.0;
      ON    DB371.DBX 1411.2;
      ON    DB376.DBX 341.2;
      JC    fui2;
// Toleranzband -3,5°C Temperatur unter der Horde
      L     DB922.DBD 1700;
      L     L#10;
      *D;
      L     L#350;	// =3,5°C
      -D;
      T     DID [AR2,P#718.0];
// Toleranzband +3,5°C Temperatur unter der Horde
      L     DB922.DBD 1700;
      L     L#10;
      *D;
      L     L#350;	// =3,5°C
      +D;
      T     DID [AR2,P#722.0];
      JU    hui2;
fui2: NOP   0;
      L     L#-10000;	// -100,00°C
      T     DID [AR2,P#714.0];
      L     L#0;	// 0,00°C
      T     DID [AR2,P#718.0];
      L     L#9900;	// 99,00°C
      T     DID [AR2,P#722.0];
      L     L#10000;	// 100,00°C
      T     DID [AR2,P#726.0];
hui2: NOP   0;
// 
//-Set Parameters---
// 
//-Call object control---
      BLD   14;
// 
//-Write outputs---
      =     L 10.0;
      L     DINO;
      T     LW 8;
      CDB;
      OPN   DI [LW 8];
      TAR2  LD 4;
      +AR2  P#676.0;
      UC    FB 19;
      LAR2  LD 4;
      CDB;
      BLD   15;
NETWORK
TITLE = Test Fault
      A     DIX [AR2,P#65.7];
      O     DIX [AR2,P#153.7];
      O     DIX [AR2,P#241.7];
//      O     #A_3191_BTE08.OutFaulted
      O     DIX [AR2,P#417.7];
      O     DIX [AR2,P#505.7];
      O     DIX [AR2,P#593.7];
      O     DIX [AR2,P#681.7];
      =     DIX [AR2,P#19.2];
NETWORK
TITLE = Test Warning
//      U     #A_3191_BTE01.OutWarning
      O     DIX [AR2,P#153.6];
      O     DIX [AR2,P#241.6];
//      O     #A_3191_BTE08.OutWarning
      O     DIX [AR2,P#417.6];
      O     DIX [AR2,P#505.6];
      O     DIX [AR2,P#593.6];
      =     DIX [AR2,P#17.6];
NETWORK
TITLE = Test Stopped
      A     DIX [AR2,P#16.2];
      A     DIX [AR2,P#19.7];
      O     DIX [AR2,P#16.0];
      AN    DIX [AR2,P#19.2];
      =     DIX [AR2,P#19.0];
NETWORK
TITLE = Test Started
      A     DIX [AR2,P#15.4];
      AN    DIX [AR2,P#19.0];
      AN    DIX [AR2,P#19.2];
      =     DIX [AR2,P#19.1];
NETWORK
TITLE = Enable Previous Group
      A     DIX [AR2,P#19.1];
      =     DIX [AR2,P#18.7];
NETWORK
TITLE = Call Methode State
//1. Make State of the group: This function use the signals:
//        Gr.VarStopped, Gr.VarStarted, Gr.VarFault
//2.Reset Commands to group: e.g.CmdFaultReset
      BLD   14;
      =     L 10.0;
      L     DINO;
      T     LW 8;
      CDB;
      OPN   DI [LW 8];
      TAR2  LD 4;
      L     2;
      T     DIW [AR2,P#0.0];
      +AR2  P#0.0;
      UC    FB 10;
      LAR2  LD 4;
      CDB;
      BLD   15;
NETWORK
TITLE = Init
      SET;
      R     DIX [AR2,P#58.2];
      R     DIX [AR2,P#58.3];
NETWORK
TITLE = Write data to group control
      A     DIX [AR2,P#17.0];
      =     DB9.DBX 483.4;
      A     DIX [AR2,P#17.2];
      =     DB9.DBX 523.4;
      A     DIX [AR2,P#17.4];
      =     DB9.DBX 563.4;
      A     DIX [AR2,P#17.6];
      =     DB9.DBX 603.4;
      A     DIX [AR2,P#18.5];
      =     DB9.DBX 643.4;
      A     DIX [AR2,P#18.2];
      =     DB9.DBX 883.4;
      A     DIX [AR2,P#18.3];
      =     DB9.DBX 843.4;
      A     DIX [AR2,P#17.5];
      =     DB9.DBX 803.4;
      A     DIX [AR2,P#18.4];
      =     DB9.DBX 923.4;
      A     DIX [AR2,P#19.3];
      =     DB9.DBX 963.4;
NETWORK
TITLE = End of block
      BE;
END_FUNCTION_BLOCK

FUNCTION_BLOCK "G285M_Code"	// FB 385
TITLE = G285M MAIN ASPIRATION 6181 - DEC1
//COPYRIGHT:    (C) 2009  BUHLER AG, CH-9240 UZWIL, SWITZERLAND
//
//PRODUCT:      WinCoS_BIW01_09
//
//TITLE:        MAIN ASPIRATION 6181 - DEC1
//                Machine group control
//                Maschinengruppensteuerung
// 
//--------------------------------------------------------------------------------
// 
//IDENT:        AUTHOR:             DEPT:                              DATE:
// 
//P01_FB385.1.0 K.Renz              CSB41                              22.Dez.2011
//             1st Release
// 
//--------------------------------------------------------------------------------
// 
//PURPOSE: 
// 
//MANUAL : 
// 
//RESTRICTIONS: 
// 
//--------------------------------------------------------------------------------
//
AUTHOR : KR
FAMILY : USW
VERSION : 9.9
VAR
  Gr : FB 10;	//Standard interface to group
  InOutValue1 : DINT ;	//Data for user
  InOutValue2 : DINT ;	//Data for user
  OutWayConflict : BOOL ;	//Data for user
  OutSelectionOk : BOOL ;	//Data for user
  CmdNewValue : BOOL ;	//Data for user
  CmdNewJob : BOOL ;	//Data for user
  OutCodeOK : BOOL ;	//Data for user
  InEndOfJob : BOOL ;	//Data for user
  staWayOk : BOOL ;	//Data for user
  EdgeStartRelease : BOOL ;	//Data for user
  USW8 : BOOL ;	//Data for user
  USW9 : BOOL ;	//Data for user
  USW10 : BOOL ;	//Data for user
  USW11 : BOOL ;	//Data for user
  USW12 : BOOL ;	//Data for user
  USW13 : BOOL ;	//Data for user
  USW14 : BOOL ;	//Data for user
  USW15 : BOOL ;	//Data for user
  A_6181_MXZ01_MA : FB 1068;	// Aspiration A
  A_6183_BSA11 : FB 14;	// DigInpCont
  A_6185_BLH01 : FB 84;	// SubType FB14: DigInpCont
  A_6186_MXZ01 : FB 12;	// Fan: Motor
END_VAR
VAR_TEMP
  tmpEnable : BOOL ;
  tmpFlag : BOOL ;
  tmpCmdNext : BOOL ;
  tmpLocal : BOOL ;
  tmpAspOk : BOOL ;
  tmpHWStop : BOOL ;
  tmpInstanzDBNo : INT ;
END_VAR
BEGIN
NETWORK
TITLE =
NETWORK
TITLE = Read command from group control
//Parameter
      SET;
      S     DB9.DBX 85.4;
      R     DB9.DBX 125.4;
      R     DB9.DBX 165.4;
      R     DB9.DBX 45.4;
      S     DB9.DBX 205.4;
      S     DIX [AR2,P#32.0];
      R     DIX [AR2,P#32.1];
      R     DIX [AR2,P#32.2];
//Command
      A     DB9.DBX 325.4;
      =     DIX [AR2,P#14.0];
      A     DB9.DBX 285.4;
      =     DIX [AR2,P#15.4];
      A     DB9.DBX 405.4;
      R     DB9.DBX 405.4;
      S     DIX [AR2,P#15.3];
      A     DB9.DBX 365.4;
      R     DB9.DBX 365.4;
      S     DIX [AR2,P#15.2];
      A     DB9.DBX 445.4;
      O     DB9.DBX 285.4;
      R     DB9.DBX 445.4;
      S     DIX [AR2,P#14.7];
      A     DB9.DBX 765.4;
      R     DB9.DBX 765.4;
      S     DIX [AR2,P#14.1];
//Init Line Number
      A     DB9.DBX 205.4;
      JCN   WE00;
      L     0;
      T     DIW [AR2,P#24.0];
WE00: NOP   0;
NETWORK
TITLE = Call Methode Control
// 1. Handle Interface PCControl      
// 2. Prepare mode --> ModePassive,ModeActive,ModeIdling      
// 3. Reset global flags of the group
      BLD   14;
      =     L 10.0;
      L     DINO;
      T     LW 8;
      CDB;
      OPN   DI [LW 8];
      TAR2  LD 4;
      L     1;
      T     DIW [AR2,P#0.0];
      +AR2  P#0.0;
      UC    FB 10;
      LAR2  LD 4;
      CDB;
      BLD   15;
NETWORK
TITLE = Restart Idling Time
      L     DIW [AR2,P#36.0];
      L     2;
      >=I;
      JC    IdTm;
      T     DIW [AR2,P#36.0];
IdTm: NOP   0;
//-Enable idling when fluidlifts and waygroups are stopped---
      A     M 50.0;
      =     M 50.0;
      CLR;
      S     DIX [AR2,P#14.2];
NETWORK
TITLE = Prepare global flags
NETWORK
TITLE = Set Pattern (Target position)
NETWORK
TITLE = Interlocking WayOk
NETWORK
TITLE = Interlocking Autostart
      CLR;
      R     DIX [AR2,P#18.4];
NETWORK
TITLE = Interlocking Enable
      A     DIX [AR2,P#14.0];
      =     DIX [AR2,P#18.0];
NETWORK
TITLE = Interlocking Next
      A     DIX [AR2,P#15.2];
      A     DIX [AR2,P#18.4];
      AN    DIX [AR2,P#19.6];
      =     #tmpCmdNext;
NETWORK
TITLE = Interlocking Local / HWStop
      A     DB50.DBX 32.7;
      =     #tmpHWStop;
      A     DIX [AR2,P#16.0];
      O     #tmpHWStop;
      =     #tmpLocal;
NETWORK
TITLE = =A-6181-MXZ01_MA : CENTRAL ASPIRATION 6181 - DEC1
      NOP   0;
//-InLocal---
      A     #tmpLocal;
      =     DIX [AR2,P#63.4];
// 
//-Interlocking---
      A     DIX [AR2,P#18.0];
      =     DIX [AR2,P#62.0];
// 
      A     #tmpCmdNext;
      S     DIX [AR2,P#63.2];
// 
      A     DIX [AR2,P#19.7];
      =     DIX [AR2,P#63.7];
// 
//-Additional commands---
      AN    DIX [AR2,P#18.0];
      =     DIX [AR2,P#62.1];
// 
      L     DIW [AR2,P#168.0];
      +     3000;
      T     DIW [AR2,P#102.0];
// 
//=Values and commands of elements===
// 
//-Read inputs of elements---
      A     I 1157.7;
      =     DIX [AR2,P#82.6];
      A     DB50.DBX 32.7;
      =     DIX [AR2,P#84.0];
      A     I 1158.0;
      =     DIX [AR2,P#116.6];
      A     DB50.DBX 32.7;
      =     DIX [AR2,P#118.0];
      A     DB50.DBX 32.7;
      =     DIX [AR2,P#152.0];
// 
//-Set Parameters---
// 
//-Call object control---
      BLD   14;
// 
//-Write outputs---
      =     L 10.0;
      L     DINO;
      T     LW 8;
      CDB;
      OPN   DI [LW 8];
      TAR2  LD 4;
      +AR2  P#60.0;
      UC    FB 1068;
      LAR2  LD 4;
      CDB;
      BLD   15;
      A     DIX [AR2,P#84.6];
      =     Q 1157.7;
      A     DIX [AR2,P#118.6];
      =     Q 1158.0;
      A     DIX [AR2,P#152.7];
      =     Q 1180.0;
      A     DIX [AR2,P#119.0];
      =     Q 1164.0;
NETWORK
TITLE = =A-6183-BSA11 : AIRLOCK 6183 - SPEED CONTROL
      NOP   0;
//-InLocal---
      A     #tmpLocal;
      =     DIX [AR2,P#355.4];
// 
//-Monitoring---
      SET;
      A     DIX [AR2,P#85.2];
      =     DIX [AR2,P#354.0];
      CLR;
      =     DIX [AR2,P#354.1];
// 
//-PreAlarm---
      CLR;
      =     DIX [AR2,P#354.2];
      CLR;
      =     DIX [AR2,P#354.3];
// 
//-Additional commands---
      AN    DIX [AR2,P#355.4];
      S     DIX [AR2,P#355.2];
// 
//-Read inputs---
      A     I 1176.3;
      =     DIX [AR2,P#354.6];
      A     DB50.DBX 32.7;
      =     DIX [AR2,P#356.0];
// 
//-Set Parameters---
// 
//-Call object control---
      BLD   14;
// 
//-Write outputs---
      =     L 10.0;
      L     DINO;
      T     LW 8;
      CDB;
      OPN   DI [LW 8];
      TAR2  LD 4;
      +AR2  P#352.0;
      UC    FB 14;
      LAR2  LD 4;
      CDB;
      BLD   15;
NETWORK
TITLE = =A-6185-BLH01 : ALARM HIGH LEVEL
      NOP   0;
//-Local---
      CLR;
      =     DIX [AR2,P#389.4];
// 
//  SET   
//   =     #A_6185_BLH01.InMonTrue
//-Read inputs---
      AN    I 1158.1;
      CLR;
      =     DIX [AR2,P#388.6];
// 
//-Set Parameters---
// 
//-Call object control---
      BLD   14;
// 
//-Write outputs---
      =     L 10.0;
      L     DINO;
      T     LW 8;
      CDB;
      OPN   DI [LW 8];
      TAR2  LD 4;
      +AR2  P#386.0;
      UC    FB 84;
      LAR2  LD 4;
      CDB;
      BLD   15;
NETWORK
TITLE = =A-6186-MXZ01 : INPUT VENTILATION 6186 - DEC1
      NOP   0;
//-InLocal---
      CLR;
      =     DIX [AR2,P#423.4];
// 
//-Interlocking---
// A     #Gr.OutEnableEl
// =     #A_6186_MXZ01.InEnableFwd
// 
      A     #tmpCmdNext;
      S     DIX [AR2,P#423.2];
// 
      A     DIX [AR2,P#19.7];
      =     DIX [AR2,P#423.7];
// 
//-Additional commands---
// 
// 
//=Values and commands of elements===
// 
//-Read inputs of elements---
//      A     "A_6186_MXZ01_I1"
      =     DIX [AR2,P#422.6];
      A     DB50.DBX 32.7;
      =     DIX [AR2,P#424.0];
// 
//-Set Parameters---
// 
//-Call object control---
      BLD   14;
// 
//-Write outputs---
      =     L 10.0;
      L     DINO;
      T     LW 8;
      CDB;
      OPN   DI [LW 8];
      TAR2  LD 4;
      +AR2  P#420.0;
      UC    FB 12;
      LAR2  LD 4;
      CDB;
      BLD   15;
NETWORK
TITLE = Test Fault
      A     DIX [AR2,P#65.4];
      O     DIX [AR2,P#357.4];
// O     #A_6185_BLH01.StFault
// O     #A_6186_MXZ01.StFault
      =     DIX [AR2,P#19.2];
NETWORK
TITLE = Test Warning
      A     DIX [AR2,P#64.0];
      =     DIX [AR2,P#17.6];
NETWORK
TITLE = Test Stopped
      A     DIX [AR2,P#65.0];
      AN    DIX [AR2,P#19.2];
      =     DIX [AR2,P#19.0];
NETWORK
TITLE = Test Started
      A(;
      A     DIX [AR2,P#65.2];
      ON    DIX [AR2,P#62.0];
      );
      AN    DIX [AR2,P#19.0];
      AN    DIX [AR2,P#19.2];
      =     DIX [AR2,P#19.1];
NETWORK
TITLE = Enable Previous Group
      A     DIX [AR2,P#19.1];
      =     DIX [AR2,P#18.7];
NETWORK
TITLE = Call Methode State
//1. Make State of the group: This function use the signals:
//        Gr.VarStopped, Gr.VarStarted, Gr.VarFault
//2.Reset Commands to group: e.g.CmdFaultReset
      BLD   14;
      =     L 10.0;
      L     DINO;
      T     LW 8;
      CDB;
      OPN   DI [LW 8];
      TAR2  LD 4;
      L     2;
      T     DIW [AR2,P#0.0];
      +AR2  P#0.0;
      UC    FB 10;
      LAR2  LD 4;
      CDB;
      BLD   15;
NETWORK
TITLE = Init
      SET;
      R     DIX [AR2,P#58.2];
      R     DIX [AR2,P#58.3];
NETWORK
TITLE = Write data to group control
      A     DIX [AR2,P#17.0];
      =     DB9.DBX 485.4;
      A     DIX [AR2,P#17.2];
      =     DB9.DBX 525.4;
      A     DIX [AR2,P#17.4];
      =     DB9.DBX 565.4;
      A     DIX [AR2,P#17.6];
      =     DB9.DBX 605.4;
      A     DIX [AR2,P#18.5];
      =     DB9.DBX 645.4;
      A     DIX [AR2,P#18.2];
      =     DB9.DBX 885.4;
      A     DIX [AR2,P#18.3];
      =     DB9.DBX 845.4;
      A     DIX [AR2,P#17.5];
      =     DB9.DBX 805.4;
      A     DIX [AR2,P#18.4];
      =     DB9.DBX 925.4;
      A     DIX [AR2,P#19.3];
      =     DB9.DBX 965.4;
NETWORK
TITLE = End of block
      BE;
END_FUNCTION_BLOCK

DATA_BLOCK "G003G"	// DB 103
TITLE = DBG003G  PLC monitoring
//COPYRIGHT:    (C) 2009  BUHLER AG, CH-9240 UZWIL, SWITZERLAND
//
//PRODUCT:      WinCoS_BIW01_09
//
//TITLE:        PLC monitoring
//                General group DB
//                Allgemeine Gruppen-DB
//
//-------------------------------------------------------------------------
//
//IDENT:        AUTHOR:             DEPT:             DATE:
//
//P01_DB103.1.0 K.Renz              CSB41             29.Sep.2009
//              1st Release
//
//-------------------------------------------------------------------------
//
//PURPOSE: 
//
//MANUAL : 
//
//RESTRICTIONS: 
//
//-------------------------------------------------------------------------
//
AUTHOR : KR
FAMILY : USW
NAME : DBG003G
VERSION : 0.0
"G003G_Code"
BEGIN
END_DATA_BLOCK

DATA_BLOCK "G269M"	// DB 369
TITLE = DBG269M  TEMPERATURE MES. KILN 1
//COPYRIGHT:    (C) 2009  BUHLER AG, CH-9240 UZWIL, SWITZERLAND
//
//PRODUCT:      WinCoS_BIW01_09
//
//TITLE:        TEMPERATURE MES. KILN 1
//                Machine group DB
//                Maschinengruppen-DB
//
//-------------------------------------------------------------------------
//
//IDENT:        AUTHOR:             DEPT:             DATE:
//
//P01_DB369.1.0 K.Renz              CSB41             30.Sep.2009
//              1st Release
//
//-------------------------------------------------------------------------
//
//PURPOSE: 
//
//MANUAL : 
//
//RESTRICTIONS: 
//
//-------------------------------------------------------------------------
//
AUTHOR : KR
FAMILY : USW
NAME : DBG269M
VERSION : 0.0
"G269M_Code"
BEGIN
END_DATA_BLOCK

DATA_BLOCK "G285M"	// DB 385
TITLE = DBG285M  MAIN ASPIRATION 6181 - DEC1
//COPYRIGHT:    (C) 2009  BUHLER AG, CH-9240 UZWIL, SWITZERLAND
//
//PRODUCT:      WinCoS_BIW01_09
//
//TITLE:        MAIN ASPIRATION 6181 - DEC1
//                Machine group DB
//                Maschinengruppen-DB
//
//-------------------------------------------------------------------------
//
//IDENT:        AUTHOR:             DEPT:             DATE:
//
//P01_DB385.1.0 K.Renz              CSB41             22.Dez.2011
//              1st Release
//
//-------------------------------------------------------------------------
//
//PURPOSE: 
//
//MANUAL : 
//
//RESTRICTIONS: 
//
//-------------------------------------------------------------------------
//
AUTHOR : KR
FAMILY : USW
NAME : DBG285M
VERSION : 0.0
"G285M_Code"
BEGIN
END_DATA_BLOCK

SYMBOL_TABLE
"G285M"	DB 385	FB 385	// Group-DB  MAIN ASPIRATION 6181 - DEC1
"G285M_Code"	FB 385	FB 385	// Group-FB  MAIN ASPIRATION 6181 - DEC1
END_SYMBOL_TABLE

